        IF nPos_Buffer = 1 GOTO pos_1;
        IF nPos_Buffer = 2 GOTO pos_2;
        IF nPos_Buffer = 3 GOTO pos_3;
        IF nPos_Buffer = 4 GOTO pos_4;
        IF nPos_Buffer = 5 GOTO pos_5;
        IF nPos_Buffer = 6 GOTO pos_6;
        IF nPos_Buffer = 7 GOTO pos_7;
        IF nPos_Buffer = 8 GOTO pos_8;
        IF nPos_Buffer = 9 GOTO pos_9;
        IF nPos_Buffer = 10 GOTO pos_10;
        IF nPos_Buffer = 11 GOTO pos_11;
        IF nPos_Buffer = 12 GOTO pos_12;
        IF nPos_Buffer = 13 GOTO pos_13;
        IF nPos_Buffer = 14 GOTO pos_14;
        IF nPos_Buffer = 15 GOTO pos_15;
        IF nPos_Buffer = 16 GOTO pos_16;
        IF nPos_Buffer = 17 GOTO pos_17;
        IF nPos_Buffer = 18 GOTO pos_18;
        IF nPos_Buffer = 19 GOTO pos_19;
        IF nPos_Buffer = 20 GOTO pos_20;
        IF nPos_Buffer = 21 GOTO pos_21;
        IF nPos_Buffer = 22 GOTO pos_22;
        IF nPos_Buffer = 23 GOTO pos_23;
        IF nPos_Buffer = 24 GOTO pos_24;
        IF nPos_Buffer = 25 GOTO pos_25;
        IF nPos_Buffer = 26 GOTO pos_26;
        IF nPos_Buffer = 27 GOTO pos_27;
        IF nPos_Buffer = 28 GOTO pos_28;
        IF nPos_Buffer = 29 GOTO pos_29;
        IF nPos_Buffer = 30 GOTO pos_30;
        IF nPos_Buffer = 31 GOTO pos_31;
        IF nPos_Buffer = 32 GOTO pos_32;
        IF nPos_Buffer = 33 GOTO pos_33;
        IF nPos_Buffer = 34 GOTO pos_34;
        IF nPos_Buffer = 35 GOTO pos_35;
        IF nPos_Buffer = 36 GOTO pos_36;
        IF nPos_Buffer = 37 GOTO pos_37;
        IF nPos_Buffer = 38 GOTO pos_38;
        IF nPos_Buffer = 39 GOTO pos_39;
        IF nPos_Buffer = 40 GOTO pos_40;
        IF nPos_Buffer = 41 GOTO pos_41;
        IF nPos_Buffer = 42 GOTO pos_42;
        IF nPos_Buffer = 43 GOTO pos_43;
        IF nPos_Buffer = 44 GOTO pos_44;
        IF nPos_Buffer = 45 GOTO pos_45;
        IF nPos_Buffer = 46 GOTO pos_46;
        IF nPos_Buffer = 47 GOTO pos_47;
        IF nPos_Buffer = 48 GOTO pos_48;
        IF nPos_Buffer = 49 GOTO pos_49;
        IF nPos_Buffer = 50 GOTO pos_50;
        IF nPos_Buffer = 51 GOTO pos_51;
        IF nPos_Buffer = 52 GOTO pos_52;
        IF nPos_Buffer = 53 GOTO pos_53;
        IF nPos_Buffer = 54 GOTO pos_54;
        IF nPos_Buffer = 55 GOTO pos_55;
        IF nPos_Buffer = 56 GOTO pos_56;
        IF nPos_Buffer = 57 GOTO pos_57;
        IF nPos_Buffer = 58 GOTO pos_58;
        IF nPos_Buffer = 59 GOTO pos_59;
        IF nPos_Buffer = 60 GOTO pos_60;
        IF nPos_Buffer = 61 GOTO pos_61;
        IF nPos_Buffer = 62 GOTO pos_62;
        IF nPos_Buffer = 63 GOTO pos_63;
        IF nPos_Buffer = 64 GOTO pos_64;
        IF nPos_Buffer = 65 GOTO pos_65;
        IF nPos_Buffer = 66 GOTO pos_66;
        IF nPos_Buffer = 67 GOTO pos_67;
        IF nPos_Buffer = 68 GOTO pos_68;
        IF nPos_Buffer = 69 GOTO pos_69;
        IF nPos_Buffer = 70 GOTO pos_70;
        IF nPos_Buffer = 71 GOTO pos_71;
        IF nPos_Buffer = 72 GOTO pos_72;
        IF nPos_Buffer = 73 GOTO pos_73;
        IF nPos_Buffer = 74 GOTO pos_74;
        IF nPos_Buffer = 75 GOTO pos_75;
        IF nPos_Buffer = 76 GOTO pos_76;
        IF nPos_Buffer = 77 GOTO pos_77;
        IF nPos_Buffer = 78 GOTO pos_78;
        IF nPos_Buffer = 79 GOTO pos_79;
        IF nPos_Buffer = 80 GOTO pos_80;
        IF nPos_Buffer = 81 GOTO pos_81;
        IF nPos_Buffer = 82 GOTO pos_82;
        IF nPos_Buffer = 83 GOTO pos_83;
        IF nPos_Buffer = 84 GOTO pos_84;
        IF nPos_Buffer = 85 GOTO pos_85;
        IF nPos_Buffer = 86 GOTO pos_86;
        IF nPos_Buffer = 87 GOTO pos_87;
        IF nPos_Buffer = 88 GOTO pos_88;
        IF nPos_Buffer = 89 GOTO pos_89;
        IF nPos_Buffer = 90 GOTO pos_90;
        IF nPos_Buffer = 91 GOTO pos_91;
        IF nPos_Buffer = 92 GOTO pos_92;
        IF nPos_Buffer = 93 GOTO pos_93;
        IF nPos_Buffer = 94 GOTO pos_94;
        IF nPos_Buffer = 95 GOTO pos_95;
        IF nPos_Buffer = 96 GOTO pos_96;
        IF nPos_Buffer = 97 GOTO pos_97;
        IF nPos_Buffer = 98 GOTO pos_98;
        IF nPos_Buffer = 99 GOTO pos_99;

    pos_1:
        !Posição 1

        !Carrega posição correspondente à familia selecionada
        IF GInput (PN_IN_Numero_Familia) = 1 THEN
            pPosição_Final_Buffer := pBuffer_Pos_1_Fam_1;
        ENDIF
        IF GInput (PN_IN_Numero_Familia) = 2 THEN
            pPosição_Final_Buffer := pBuffer_Pos_1_Fam_2;
        ENDIF
        IF GInput (PN_IN_Numero_Familia) = 3 THEN
            pPosição_Final_Buffer := pBuffer_Pos_1_Fam_3;
        ENDIF
        IF GInput (PN_IN_Numero_Familia) = 4 THEN
            pPosição_Final_Buffer := pBuffer_Pos_1_Fam_4;
        ENDIF

        GOTO verifica_passo;

    pos_2:
        !Posição 2

        !Carrega posição correspondente à familia selecionada
        IF GInput (PN_IN_Numero_Familia) = 1 THEN
            pPosição_Final_Buffer := pBuffer_Pos_2_Fam_1;
        ENDIF
        IF GInput (PN_IN_Numero_Familia) = 2 THEN
            pPosição_Final_Buffer := pBuffer_Pos_2_Fam_2;
        ENDIF
        IF GInput (PN_IN_Numero_Familia) = 3 THEN
            pPosição_Final_Buffer := pBuffer_Pos_2_Fam_3;
        ENDIF
        IF GInput (PN_IN_Numero_Familia) = 4 THEN
            pPosição_Final_Buffer := pBuffer_Pos_2_Fam_4;
        ENDIF

        GOTO verifica_passo;

    pos_3:
        !Posição 3

        !Carrega posição correspondente à familia selecionada
        IF GInput (PN_IN_Numero_Familia) = 1 THEN
            pPosição_Final_Buffer := pBuffer_Pos_3_Fam_1;
        ENDIF
        IF GInput (PN_IN_Numero_Familia) = 2 THEN
            pPosição_Final_Buffer := pBuffer_Pos_3_Fam_2;
        ENDIF
        IF GInput (PN_IN_Numero_Familia) = 3 THEN
            pPosição_Final_Buffer := pBuffer_Pos_3_Fam_3;
        ENDIF
        IF GInput (PN_IN_Numero_Familia) = 4 THEN
            pPosição_Final_Buffer := pBuffer_Pos_3_Fam_4;
        ENDIF

        GOTO verifica_passo;

    pos_4:
        !Posição 4

        !Carrega posição correspondente à familia selecionada
        IF GInput (PN_IN_Numero_Familia) = 1 THEN
            pPosição_Final_Buffer := pBuffer_Pos_4_Fam_1;
        ENDIF
        IF GInput (PN_IN_Numero_Familia) = 2 THEN
            pPosição_Final_Buffer := pBuffer_Pos_4_Fam_2;
        ENDIF
        IF GInput (PN_IN_Numero_Familia) = 3 THEN
            pPosição_Final_Buffer := pBuffer_Pos_4_Fam_3;
        ENDIF
        IF GInput (PN_IN_Numero_Familia) = 4 THEN
            pPosição_Final_Buffer := pBuffer_Pos_4_Fam_4;
        ENDIF

        GOTO verifica_passo;

    pos_5:
        !Posição 5

        !Carrega posição correspondente à familia selecionada
        IF GInput (PN_IN_Numero_Familia) = 1 THEN
            pPosição_Final_Buffer := pBuffer_Pos_5_Fam_1;
        ENDIF
        IF GInput (PN_IN_Numero_Familia) = 2 THEN
            pPosição_Final_Buffer := pBuffer_Pos_5_Fam_2;
        ENDIF
        IF GInput (PN_IN_Numero_Familia) = 3 THEN
            pPosição_Final_Buffer := pBuffer_Pos_5_Fam_3;
        ENDIF
        IF GInput (PN_IN_Numero_Familia) = 4 THEN
            pPosição_Final_Buffer := pBuffer_Pos_5_Fam_4;
        ENDIF

        GOTO verifica_passo;

    pos_6:
        !Posição 6

        !Carrega posição correspondente à familia selecionada
        IF GInput (PN_IN_Numero_Familia) = 1 THEN
            pPosição_Final_Buffer := pBuffer_Pos_6_Fam_1;
        ENDIF
        IF GInput (PN_IN_Numero_Familia) = 2 THEN
            pPosição_Final_Buffer := pBuffer_Pos_6_Fam_2;
        ENDIF
        IF GInput (PN_IN_Numero_Familia) = 3 THEN
            pPosição_Final_Buffer := pBuffer_Pos_6_Fam_3;
        ENDIF
        IF GInput (PN_IN_Numero_Familia) = 4 THEN
            pPosição_Final_Buffer := pBuffer_Pos_6_Fam_4;
        ENDIF

        GOTO verifica_passo;

    pos_7:
        !Posição 7

        !Carrega posição correspondente à familia selecionada
        IF GInput (PN_IN_Numero_Familia) = 1 THEN
            pPosição_Final_Buffer := pBuffer_Pos_7_Fam_1;
        ENDIF
        IF GInput (PN_IN_Numero_Familia) = 2 THEN
            pPosição_Final_Buffer := pBuffer_Pos_7_Fam_2;
        ENDIF
        IF GInput (PN_IN_Numero_Familia) = 3 THEN
            pPosição_Final_Buffer := pBuffer_Pos_7_Fam_3;
        ENDIF
        IF GInput (PN_IN_Numero_Familia) = 4 THEN
            pPosição_Final_Buffer := pBuffer_Pos_7_Fam_4;
        ENDIF

        GOTO verifica_passo;

    pos_8:
        !Posição 8

        !Carrega posição correspondente à familia selecionada
        IF GInput (PN_IN_Numero_Familia) = 1 THEN
            pPosição_Final_Buffer := pBuffer_Pos_8_Fam_1;
        ENDIF
        IF GInput (PN_IN_Numero_Familia) = 2 THEN
            pPosição_Final_Buffer := pBuffer_Pos_8_Fam_2;
        ENDIF
        IF GInput (PN_IN_Numero_Familia) = 3 THEN
            pPosição_Final_Buffer := pBuffer_Pos_8_Fam_3;
        ENDIF
        IF GInput (PN_IN_Numero_Familia) = 4 THEN
            pPosição_Final_Buffer := pBuffer_Pos_8_Fam_4;
        ENDIF

        GOTO verifica_passo;

    pos_9:
        !Posição 9

        !Carrega posição correspondente à familia selecionada
        IF GInput (PN_IN_Numero_Familia) = 1 THEN
            pPosição_Final_Buffer := pBuffer_Pos_9_Fam_1;
        ENDIF
        IF GInput (PN_IN_Numero_Familia) = 2 THEN
            pPosição_Final_Buffer := pBuffer_Pos_9_Fam_2;
        ENDIF
        IF GInput (PN_IN_Numero_Familia) = 3 THEN
            pPosição_Final_Buffer := pBuffer_Pos_9_Fam_3;
        ENDIF
        IF GInput (PN_IN_Numero_Familia) = 4 THEN
            pPosição_Final_Buffer := pBuffer_Pos_9_Fam_4;
        ENDIF

        GOTO verifica_passo;

    pos_10:
        !Posição 10

        !Carrega posição correspondente à familia selecionada
        IF GInput (PN_IN_Numero_Familia) = 1 THEN
            pPosição_Final_Buffer := pBuffer_Pos_10_Fam_1;
        ENDIF
        IF GInput (PN_IN_Numero_Familia) = 2 THEN
            pPosição_Final_Buffer := pBuffer_Pos_10_Fam_2;
        ENDIF
        IF GInput (PN_IN_Numero_Familia) = 3 THEN
            pPosição_Final_Buffer := pBuffer_Pos_10_Fam_3;
        ENDIF
        IF GInput (PN_IN_Numero_Familia) = 4 THEN
            pPosição_Final_Buffer := pBuffer_Pos_10_Fam_4;
        ENDIF

        GOTO verifica_passo;

    pos_11:
        !Posição 11

        !Carrega posição correspondente à familia selecionada
        IF GInput (PN_IN_Numero_Familia) = 1 THEN
            pPosição_Final_Buffer := pBuffer_Pos_11_Fam_1;
        ENDIF
        IF GInput (PN_IN_Numero_Familia) = 2 THEN
            pPosição_Final_Buffer := pBuffer_Pos_11_Fam_2;
        ENDIF
        IF GInput (PN_IN_Numero_Familia) = 3 THEN
            pPosição_Final_Buffer := pBuffer_Pos_11_Fam_3;
        ENDIF
        IF GInput (PN_IN_Numero_Familia) = 4 THEN
            pPosição_Final_Buffer := pBuffer_Pos_11_Fam_4;
        ENDIF

        GOTO verifica_passo;

    pos_12:
        !Posição 12

        !Carrega posição correspondente à familia selecionada
        IF GInput (PN_IN_Numero_Familia) = 1 THEN
            pPosição_Final_Buffer := pBuffer_Pos_12_Fam_1;
        ENDIF
        IF GInput (PN_IN_Numero_Familia) = 2 THEN
            pPosição_Final_Buffer := pBuffer_Pos_12_Fam_2;
        ENDIF
        IF GInput (PN_IN_Numero_Familia) = 3 THEN
            pPosição_Final_Buffer := pBuffer_Pos_12_Fam_3;
        ENDIF
        IF GInput (PN_IN_Numero_Familia) = 4 THEN
            pPosição_Final_Buffer := pBuffer_Pos_12_Fam_4;
        ENDIF

        GOTO verifica_passo;

    pos_13:
        !Posição 13

        !Carrega posição correspondente à familia selecionada
        IF GInput (PN_IN_Numero_Familia) = 1 THEN
            pPosição_Final_Buffer := pBuffer_Pos_13_Fam_1;
        ENDIF
        IF GInput (PN_IN_Numero_Familia) = 2 THEN
            pPosição_Final_Buffer := pBuffer_Pos_13_Fam_2;
        ENDIF
        IF GInput (PN_IN_Numero_Familia) = 3 THEN
            pPosição_Final_Buffer := pBuffer_Pos_13_Fam_3;
        ENDIF
        IF GInput (PN_IN_Numero_Familia) = 4 THEN
            pPosição_Final_Buffer := pBuffer_Pos_13_Fam_4;
        ENDIF

        GOTO verifica_passo;

    pos_14:
        !Posição 14

        !Carrega posição correspondente à familia selecionada
        IF GInput (PN_IN_Numero_Familia) = 1 THEN
            pPosição_Final_Buffer := pBuffer_Pos_14_Fam_1;
        ENDIF
        IF GInput (PN_IN_Numero_Familia) = 2 THEN
            pPosição_Final_Buffer := pBuffer_Pos_14_Fam_2;
        ENDIF
        IF GInput (PN_IN_Numero_Familia) = 3 THEN
            pPosição_Final_Buffer := pBuffer_Pos_14_Fam_3;
        ENDIF
        IF GInput (PN_IN_Numero_Familia) = 4 THEN
            pPosição_Final_Buffer := pBuffer_Pos_14_Fam_4;
        ENDIF

        GOTO verifica_passo;

    pos_15:
        !Posição 15

        !Carrega posição correspondente à familia selecionada
        IF GInput (PN_IN_Numero_Familia) = 1 THEN
            pPosição_Final_Buffer := pBuffer_Pos_15_Fam_1;
        ENDIF
        IF GInput (PN_IN_Numero_Familia) = 2 THEN
            pPosição_Final_Buffer := pBuffer_Pos_15_Fam_2;
        ENDIF
        IF GInput (PN_IN_Numero_Familia) = 3 THEN
            pPosição_Final_Buffer := pBuffer_Pos_15_Fam_3;
        ENDIF
        IF GInput (PN_IN_Numero_Familia) = 4 THEN
            pPosição_Final_Buffer := pBuffer_Pos_15_Fam_4;
        ENDIF

        GOTO verifica_passo;

    pos_16:
        !Posição 16

        !Carrega posição correspondente à familia selecionada
        IF GInput (PN_IN_Numero_Familia) = 1 THEN
            pPosição_Final_Buffer := pBuffer_Pos_16_Fam_1;
        ENDIF
        IF GInput (PN_IN_Numero_Familia) = 2 THEN
            pPosição_Final_Buffer := pBuffer_Pos_16_Fam_2;
        ENDIF
        IF GInput (PN_IN_Numero_Familia) = 3 THEN
            pPosição_Final_Buffer := pBuffer_Pos_16_Fam_3;
        ENDIF
        IF GInput (PN_IN_Numero_Familia) = 4 THEN
            pPosição_Final_Buffer := pBuffer_Pos_16_Fam_4;
        ENDIF

        GOTO verifica_passo;

    pos_17:
        !Posição 17

        !Carrega posição correspondente à familia selecionada
        IF GInput (PN_IN_Numero_Familia) = 1 THEN
            pPosição_Final_Buffer := pBuffer_Pos_17_Fam_1;
        ENDIF
        IF GInput (PN_IN_Numero_Familia) = 2 THEN
            pPosição_Final_Buffer := pBuffer_Pos_17_Fam_2;
        ENDIF
        IF GInput (PN_IN_Numero_Familia) = 3 THEN
            pPosição_Final_Buffer := pBuffer_Pos_17_Fam_3;
        ENDIF
        IF GInput (PN_IN_Numero_Familia) = 4 THEN
            pPosição_Final_Buffer := pBuffer_Pos_17_Fam_4;
        ENDIF

        GOTO verifica_passo;

    pos_18:
        !Posição 18

        !Carrega posição correspondente à familia selecionada
        IF GInput (PN_IN_Numero_Familia) = 1 THEN
            pPosição_Final_Buffer := pBuffer_Pos_18_Fam_1;
        ENDIF
        IF GInput (PN_IN_Numero_Familia) = 2 THEN
            pPosição_Final_Buffer := pBuffer_Pos_18_Fam_2;
        ENDIF
        IF GInput (PN_IN_Numero_Familia) = 3 THEN
            pPosição_Final_Buffer := pBuffer_Pos_18_Fam_3;
        ENDIF
        IF GInput (PN_IN_Numero_Familia) = 4 THEN
            pPosição_Final_Buffer := pBuffer_Pos_18_Fam_4;
        ENDIF

        GOTO verifica_passo;

    pos_19:
        !Posição 19

        !Carrega posição correspondente à familia selecionada
        IF GInput (PN_IN_Numero_Familia) = 1 THEN
            pPosição_Final_Buffer := pBuffer_Pos_19_Fam_1;
        ENDIF
        IF GInput (PN_IN_Numero_Familia) = 2 THEN
            pPosição_Final_Buffer := pBuffer_Pos_19_Fam_2;
        ENDIF
        IF GInput (PN_IN_Numero_Familia) = 3 THEN
            pPosição_Final_Buffer := pBuffer_Pos_19_Fam_3;
        ENDIF
        IF GInput (PN_IN_Numero_Familia) = 4 THEN
            pPosição_Final_Buffer := pBuffer_Pos_19_Fam_4;
        ENDIF

        GOTO verifica_passo;

    pos_20:
        !Posição 20

        !Carrega posição correspondente à familia selecionada
        IF GInput (PN_IN_Numero_Familia) = 1 THEN
            pPosição_Final_Buffer := pBuffer_Pos_20_Fam_1;
        ENDIF
        IF GInput (PN_IN_Numero_Familia) = 2 THEN
            pPosição_Final_Buffer := pBuffer_Pos_20_Fam_2;
        ENDIF
        IF GInput (PN_IN_Numero_Familia) = 3 THEN
            pPosição_Final_Buffer := pBuffer_Pos_20_Fam_3;
        ENDIF
        IF GInput (PN_IN_Numero_Familia) = 4 THEN
            pPosição_Final_Buffer := pBuffer_Pos_20_Fam_4;
        ENDIF

        GOTO verifica_passo;

    pos_21:
        !Posição 21

        !Carrega posição correspondente à familia selecionada
        IF GInput (PN_IN_Numero_Familia) = 1 THEN
            pPosição_Final_Buffer := pBuffer_Pos_21_Fam_1;
        ENDIF
        IF GInput (PN_IN_Numero_Familia) = 2 THEN
            pPosição_Final_Buffer := pBuffer_Pos_21_Fam_2;
        ENDIF
        IF GInput (PN_IN_Numero_Familia) = 3 THEN
            pPosição_Final_Buffer := pBuffer_Pos_21_Fam_3;
        ENDIF
        IF GInput (PN_IN_Numero_Familia) = 4 THEN
            pPosição_Final_Buffer := pBuffer_Pos_21_Fam_4;
        ENDIF

        GOTO verifica_passo;

    pos_22:
        !Posição 22

        !Carrega posição correspondente à familia selecionada
        IF GInput (PN_IN_Numero_Familia) = 1 THEN
            pPosição_Final_Buffer := pBuffer_Pos_22_Fam_1;
        ENDIF
        IF GInput (PN_IN_Numero_Familia) = 2 THEN
            pPosição_Final_Buffer := pBuffer_Pos_22_Fam_2;
        ENDIF
        IF GInput (PN_IN_Numero_Familia) = 3 THEN
            pPosição_Final_Buffer := pBuffer_Pos_22_Fam_3;
        ENDIF
        IF GInput (PN_IN_Numero_Familia) = 4 THEN
            pPosição_Final_Buffer := pBuffer_Pos_22_Fam_4;
        ENDIF

        GOTO verifica_passo;

    pos_23:
        !Posição 23

        !Carrega posição correspondente à familia selecionada
        IF GInput (PN_IN_Numero_Familia) = 1 THEN
            pPosição_Final_Buffer := pBuffer_Pos_23_Fam_1;
        ENDIF
        IF GInput (PN_IN_Numero_Familia) = 2 THEN
            pPosição_Final_Buffer := pBuffer_Pos_23_Fam_2;
        ENDIF
        IF GInput (PN_IN_Numero_Familia) = 3 THEN
            pPosição_Final_Buffer := pBuffer_Pos_23_Fam_3;
        ENDIF
        IF GInput (PN_IN_Numero_Familia) = 4 THEN
            pPosição_Final_Buffer := pBuffer_Pos_23_Fam_4;
        ENDIF

        GOTO verifica_passo;

    pos_24:
        !Posição 24

        !Carrega posição correspondente à familia selecionada
        IF GInput (PN_IN_Numero_Familia) = 1 THEN
            pPosição_Final_Buffer := pBuffer_Pos_24_Fam_1;
        ENDIF
        IF GInput (PN_IN_Numero_Familia) = 2 THEN
            pPosição_Final_Buffer := pBuffer_Pos_24_Fam_2;
        ENDIF
        IF GInput (PN_IN_Numero_Familia) = 3 THEN
            pPosição_Final_Buffer := pBuffer_Pos_24_Fam_3;
        ENDIF
        IF GInput (PN_IN_Numero_Familia) = 4 THEN
            pPosição_Final_Buffer := pBuffer_Pos_24_Fam_4;
        ENDIF

        GOTO verifica_passo;

    pos_25:
        !Posição 25

        !Carrega posição correspondente à familia selecionada
        IF GInput (PN_IN_Numero_Familia) = 1 THEN
            pPosição_Final_Buffer := pBuffer_Pos_25_Fam_1;
        ENDIF
        IF GInput (PN_IN_Numero_Familia) = 2 THEN
            pPosição_Final_Buffer := pBuffer_Pos_25_Fam_2;
        ENDIF
        IF GInput (PN_IN_Numero_Familia) = 3 THEN
            pPosição_Final_Buffer := pBuffer_Pos_25_Fam_3;
        ENDIF
        IF GInput (PN_IN_Numero_Familia) = 4 THEN
            pPosição_Final_Buffer := pBuffer_Pos_25_Fam_4;
        ENDIF

        GOTO verifica_passo;

    pos_26:
        !Posição 26

        !Carrega posição correspondente à familia selecionada
        IF GInput (PN_IN_Numero_Familia) = 1 THEN
            pPosição_Final_Buffer := pBuffer_Pos_26_Fam_1;
        ENDIF
        IF GInput (PN_IN_Numero_Familia) = 2 THEN
            pPosição_Final_Buffer := pBuffer_Pos_26_Fam_2;
        ENDIF
        IF GInput (PN_IN_Numero_Familia) = 3 THEN
            pPosição_Final_Buffer := pBuffer_Pos_26_Fam_3;
        ENDIF
        IF GInput (PN_IN_Numero_Familia) = 4 THEN
            pPosição_Final_Buffer := pBuffer_Pos_26_Fam_4;
        ENDIF

        GOTO verifica_passo;

    pos_27:
        !Posição 27

        !Carrega posição correspondente à familia selecionada
        IF GInput (PN_IN_Numero_Familia) = 1 THEN
            pPosição_Final_Buffer := pBuffer_Pos_27_Fam_1;
        ENDIF
        IF GInput (PN_IN_Numero_Familia) = 2 THEN
            pPosição_Final_Buffer := pBuffer_Pos_27_Fam_2;
        ENDIF
        IF GInput (PN_IN_Numero_Familia) = 3 THEN
            pPosição_Final_Buffer := pBuffer_Pos_27_Fam_3;
        ENDIF
        IF GInput (PN_IN_Numero_Familia) = 4 THEN
            pPosição_Final_Buffer := pBuffer_Pos_27_Fam_4;
        ENDIF

        GOTO verifica_passo;

    pos_28:
        !Posição 28

        !Carrega posição correspondente à familia selecionada
        IF GInput (PN_IN_Numero_Familia) = 1 THEN
            pPosição_Final_Buffer := pBuffer_Pos_28_Fam_1;
        ENDIF
        IF GInput (PN_IN_Numero_Familia) = 2 THEN
            pPosição_Final_Buffer := pBuffer_Pos_28_Fam_2;
        ENDIF
        IF GInput (PN_IN_Numero_Familia) = 3 THEN
            pPosição_Final_Buffer := pBuffer_Pos_28_Fam_3;
        ENDIF
        IF GInput (PN_IN_Numero_Familia) = 4 THEN
            pPosição_Final_Buffer := pBuffer_Pos_28_Fam_4;
        ENDIF

        GOTO verifica_passo;

    pos_29:
        !Posição 29

        !Carrega posição correspondente à familia selecionada
        IF GInput (PN_IN_Numero_Familia) = 1 THEN
            pPosição_Final_Buffer := pBuffer_Pos_29_Fam_1;
        ENDIF
        IF GInput (PN_IN_Numero_Familia) = 2 THEN
            pPosição_Final_Buffer := pBuffer_Pos_29_Fam_2;
        ENDIF
        IF GInput (PN_IN_Numero_Familia) = 3 THEN
            pPosição_Final_Buffer := pBuffer_Pos_29_Fam_3;
        ENDIF
        IF GInput (PN_IN_Numero_Familia) = 4 THEN
            pPosição_Final_Buffer := pBuffer_Pos_29_Fam_4;
        ENDIF

        GOTO verifica_passo;

    pos_30:
        !Posição 30

        !Carrega posição correspondente à familia selecionada
        IF GInput (PN_IN_Numero_Familia) = 1 THEN
            pPosição_Final_Buffer := pBuffer_Pos_30_Fam_1;
        ENDIF
        IF GInput (PN_IN_Numero_Familia) = 2 THEN
            pPosição_Final_Buffer := pBuffer_Pos_30_Fam_2;
        ENDIF
        IF GInput (PN_IN_Numero_Familia) = 3 THEN
            pPosição_Final_Buffer := pBuffer_Pos_30_Fam_3;
        ENDIF
        IF GInput (PN_IN_Numero_Familia) = 4 THEN
            pPosição_Final_Buffer := pBuffer_Pos_30_Fam_4;
        ENDIF

        GOTO verifica_passo;

    pos_31:
        !Posição 31

        !Carrega posição correspondente à familia selecionada
        IF GInput (PN_IN_Numero_Familia) = 1 THEN
            pPosição_Final_Buffer := pBuffer_Pos_31_Fam_1;
        ENDIF
        IF GInput (PN_IN_Numero_Familia) = 2 THEN
            pPosição_Final_Buffer := pBuffer_Pos_31_Fam_2;
        ENDIF
        IF GInput (PN_IN_Numero_Familia) = 3 THEN
            pPosição_Final_Buffer := pBuffer_Pos_31_Fam_3;
        ENDIF
        IF GInput (PN_IN_Numero_Familia) = 4 THEN
            pPosição_Final_Buffer := pBuffer_Pos_31_Fam_4;
        ENDIF

        GOTO verifica_passo;

    pos_32:
        !Posição 32

        !Carrega posição correspondente à familia selecionada
        IF GInput (PN_IN_Numero_Familia) = 1 THEN
            pPosição_Final_Buffer := pBuffer_Pos_32_Fam_1;
        ENDIF
        IF GInput (PN_IN_Numero_Familia) = 2 THEN
            pPosição_Final_Buffer := pBuffer_Pos_32_Fam_2;
        ENDIF
        IF GInput (PN_IN_Numero_Familia) = 3 THEN
            pPosição_Final_Buffer := pBuffer_Pos_32_Fam_3;
        ENDIF
        IF GInput (PN_IN_Numero_Familia) = 4 THEN
            pPosição_Final_Buffer := pBuffer_Pos_32_Fam_4;
        ENDIF

        GOTO verifica_passo;

    pos_33:
        !Posição 33

        !Carrega posição correspondente à familia selecionada
        IF GInput (PN_IN_Numero_Familia) = 1 THEN
            pPosição_Final_Buffer := pBuffer_Pos_33_Fam_1;
        ENDIF
        IF GInput (PN_IN_Numero_Familia) = 2 THEN
            pPosição_Final_Buffer := pBuffer_Pos_33_Fam_2;
        ENDIF
        IF GInput (PN_IN_Numero_Familia) = 3 THEN
            pPosição_Final_Buffer := pBuffer_Pos_33_Fam_3;
        ENDIF
        IF GInput (PN_IN_Numero_Familia) = 4 THEN
            pPosição_Final_Buffer := pBuffer_Pos_33_Fam_4;
        ENDIF

        GOTO verifica_passo;

    pos_34:
        !Posição 34

        !Carrega posição correspondente à familia selecionada
        IF GInput (PN_IN_Numero_Familia) = 1 THEN
            pPosição_Final_Buffer := pBuffer_Pos_34_Fam_1;
        ENDIF
        IF GInput (PN_IN_Numero_Familia) = 2 THEN
            pPosição_Final_Buffer := pBuffer_Pos_34_Fam_2;
        ENDIF
        IF GInput (PN_IN_Numero_Familia) = 3 THEN
            pPosição_Final_Buffer := pBuffer_Pos_34_Fam_3;
        ENDIF
        IF GInput (PN_IN_Numero_Familia) = 4 THEN
            pPosição_Final_Buffer := pBuffer_Pos_34_Fam_4;
        ENDIF

        GOTO verifica_passo;

    pos_35:
        !Posição 35

        !Carrega posição correspondente à familia selecionada
        IF GInput (PN_IN_Numero_Familia) = 1 THEN
            pPosição_Final_Buffer := pBuffer_Pos_35_Fam_1;
        ENDIF
        IF GInput (PN_IN_Numero_Familia) = 2 THEN
            pPosição_Final_Buffer := pBuffer_Pos_35_Fam_2;
        ENDIF
        IF GInput (PN_IN_Numero_Familia) = 3 THEN
            pPosição_Final_Buffer := pBuffer_Pos_35_Fam_3;
        ENDIF
        IF GInput (PN_IN_Numero_Familia) = 4 THEN
            pPosição_Final_Buffer := pBuffer_Pos_35_Fam_4;
        ENDIF

        GOTO verifica_passo;

    pos_36:
        !Posição 36

        !Carrega posição correspondente à familia selecionada
        IF GInput (PN_IN_Numero_Familia) = 1 THEN
            pPosição_Final_Buffer := pBuffer_Pos_36_Fam_1;
        ENDIF
        IF GInput (PN_IN_Numero_Familia) = 2 THEN
            pPosição_Final_Buffer := pBuffer_Pos_36_Fam_2;
        ENDIF
        IF GInput (PN_IN_Numero_Familia) = 3 THEN
            pPosição_Final_Buffer := pBuffer_Pos_36_Fam_3;
        ENDIF
        IF GInput (PN_IN_Numero_Familia) = 4 THEN
            pPosição_Final_Buffer := pBuffer_Pos_36_Fam_4;
        ENDIF

        GOTO verifica_passo;

    pos_37:
        !Posição 37

        !Carrega posição correspondente à familia selecionada
        IF GInput (PN_IN_Numero_Familia) = 1 THEN
            pPosição_Final_Buffer := pBuffer_Pos_37_Fam_1;
        ENDIF
        IF GInput (PN_IN_Numero_Familia) = 2 THEN
            pPosição_Final_Buffer := pBuffer_Pos_37_Fam_2;
        ENDIF
        IF GInput (PN_IN_Numero_Familia) = 3 THEN
            pPosição_Final_Buffer := pBuffer_Pos_37_Fam_3;
        ENDIF
        IF GInput (PN_IN_Numero_Familia) = 4 THEN
            pPosição_Final_Buffer := pBuffer_Pos_37_Fam_4;
        ENDIF

        GOTO verifica_passo;

    pos_38:
        !Posição 38

        !Carrega posição correspondente à familia selecionada
        IF GInput (PN_IN_Numero_Familia) = 1 THEN
            pPosição_Final_Buffer := pBuffer_Pos_38_Fam_1;
        ENDIF
        IF GInput (PN_IN_Numero_Familia) = 2 THEN
            pPosição_Final_Buffer := pBuffer_Pos_38_Fam_2;
        ENDIF
        IF GInput (PN_IN_Numero_Familia) = 3 THEN
            pPosição_Final_Buffer := pBuffer_Pos_38_Fam_3;
        ENDIF
        IF GInput (PN_IN_Numero_Familia) = 4 THEN
            pPosição_Final_Buffer := pBuffer_Pos_38_Fam_4;
        ENDIF

        GOTO verifica_passo;

    pos_39:
        !Posição 39

        !Carrega posição correspondente à familia selecionada
        IF GInput (PN_IN_Numero_Familia) = 1 THEN
            pPosição_Final_Buffer := pBuffer_Pos_39_Fam_1;
        ENDIF
        IF GInput (PN_IN_Numero_Familia) = 2 THEN
            pPosição_Final_Buffer := pBuffer_Pos_39_Fam_2;
        ENDIF
        IF GInput (PN_IN_Numero_Familia) = 3 THEN
            pPosição_Final_Buffer := pBuffer_Pos_39_Fam_3;
        ENDIF
        IF GInput (PN_IN_Numero_Familia) = 4 THEN
            pPosição_Final_Buffer := pBuffer_Pos_39_Fam_4;
        ENDIF

        GOTO verifica_passo;

    pos_40:
        !Posição 40

        !Carrega posição correspondente à familia selecionada
        IF GInput (PN_IN_Numero_Familia) = 1 THEN
            pPosição_Final_Buffer := pBuffer_Pos_40_Fam_1;
        ENDIF
        IF GInput (PN_IN_Numero_Familia) = 2 THEN
            pPosição_Final_Buffer := pBuffer_Pos_40_Fam_2;
        ENDIF
        IF GInput (PN_IN_Numero_Familia) = 3 THEN
            pPosição_Final_Buffer := pBuffer_Pos_40_Fam_3;
        ENDIF
        IF GInput (PN_IN_Numero_Familia) = 4 THEN
            pPosição_Final_Buffer := pBuffer_Pos_40_Fam_4;
        ENDIF

        GOTO verifica_passo;

    pos_41:
        !Posição 41

        !Carrega posição correspondente à familia selecionada
        IF GInput (PN_IN_Numero_Familia) = 1 THEN
            pPosição_Final_Buffer := pBuffer_Pos_41_Fam_1;
        ENDIF
        IF GInput (PN_IN_Numero_Familia) = 2 THEN
            pPosição_Final_Buffer := pBuffer_Pos_41_Fam_2;
        ENDIF
        IF GInput (PN_IN_Numero_Familia) = 3 THEN
            pPosição_Final_Buffer := pBuffer_Pos_41_Fam_3;
        ENDIF
        IF GInput (PN_IN_Numero_Familia) = 4 THEN
            pPosição_Final_Buffer := pBuffer_Pos_41_Fam_4;
        ENDIF

        GOTO verifica_passo;

    pos_42:
        !Posição 42

        !Carrega posição correspondente à familia selecionada
        IF GInput (PN_IN_Numero_Familia) = 1 THEN
            pPosição_Final_Buffer := pBuffer_Pos_42_Fam_1;
        ENDIF
        IF GInput (PN_IN_Numero_Familia) = 2 THEN
            pPosição_Final_Buffer := pBuffer_Pos_42_Fam_2;
        ENDIF
        IF GInput (PN_IN_Numero_Familia) = 3 THEN
            pPosição_Final_Buffer := pBuffer_Pos_42_Fam_3;
        ENDIF
        IF GInput (PN_IN_Numero_Familia) = 4 THEN
            pPosição_Final_Buffer := pBuffer_Pos_42_Fam_4;
        ENDIF

        GOTO verifica_passo;

    pos_43:
        !Posição 43

        !Carrega posição correspondente à familia selecionada
        IF GInput (PN_IN_Numero_Familia) = 1 THEN
            pPosição_Final_Buffer := pBuffer_Pos_43_Fam_1;
        ENDIF
        IF GInput (PN_IN_Numero_Familia) = 2 THEN
            pPosição_Final_Buffer := pBuffer_Pos_43_Fam_2;
        ENDIF
        IF GInput (PN_IN_Numero_Familia) = 3 THEN
            pPosição_Final_Buffer := pBuffer_Pos_43_Fam_3;
        ENDIF
        IF GInput (PN_IN_Numero_Familia) = 4 THEN
            pPosição_Final_Buffer := pBuffer_Pos_43_Fam_4;
        ENDIF

        GOTO verifica_passo;

    pos_44:
        !Posição 44

        !Carrega posição correspondente à familia selecionada
        IF GInput (PN_IN_Numero_Familia) = 1 THEN
            pPosição_Final_Buffer := pBuffer_Pos_44_Fam_1;
        ENDIF
        IF GInput (PN_IN_Numero_Familia) = 2 THEN
            pPosição_Final_Buffer := pBuffer_Pos_44_Fam_2;
        ENDIF
        IF GInput (PN_IN_Numero_Familia) = 3 THEN
            pPosição_Final_Buffer := pBuffer_Pos_44_Fam_3;
        ENDIF
        IF GInput (PN_IN_Numero_Familia) = 4 THEN
            pPosição_Final_Buffer := pBuffer_Pos_44_Fam_4;
        ENDIF

        GOTO verifica_passo;

    pos_45:
        !Posição 45

        !Carrega posição correspondente à familia selecionada
        IF GInput (PN_IN_Numero_Familia) = 1 THEN
            pPosição_Final_Buffer := pBuffer_Pos_45_Fam_1;
        ENDIF
        IF GInput (PN_IN_Numero_Familia) = 2 THEN
            pPosição_Final_Buffer := pBuffer_Pos_45_Fam_2;
        ENDIF
        IF GInput (PN_IN_Numero_Familia) = 3 THEN
            pPosição_Final_Buffer := pBuffer_Pos_45_Fam_3;
        ENDIF
        IF GInput (PN_IN_Numero_Familia) = 4 THEN
            pPosição_Final_Buffer := pBuffer_Pos_45_Fam_4;
        ENDIF

        GOTO verifica_passo;

    pos_46:
        !Posição 46

        !Carrega posição correspondente à familia selecionada
        IF GInput (PN_IN_Numero_Familia) = 1 THEN
            pPosição_Final_Buffer := pBuffer_Pos_46_Fam_1;
        ENDIF
        IF GInput (PN_IN_Numero_Familia) = 2 THEN
            pPosição_Final_Buffer := pBuffer_Pos_46_Fam_2;
        ENDIF
        IF GInput (PN_IN_Numero_Familia) = 3 THEN
            pPosição_Final_Buffer := pBuffer_Pos_46_Fam_3;
        ENDIF
        IF GInput (PN_IN_Numero_Familia) = 4 THEN
            pPosição_Final_Buffer := pBuffer_Pos_46_Fam_4;
        ENDIF

        GOTO verifica_passo;

    pos_47:
        !Posição 47

        !Carrega posição correspondente à familia selecionada
        IF GInput (PN_IN_Numero_Familia) = 1 THEN
            pPosição_Final_Buffer := pBuffer_Pos_47_Fam_1;
        ENDIF
        IF GInput (PN_IN_Numero_Familia) = 2 THEN
            pPosição_Final_Buffer := pBuffer_Pos_47_Fam_2;
        ENDIF
        IF GInput (PN_IN_Numero_Familia) = 3 THEN
            pPosição_Final_Buffer := pBuffer_Pos_47_Fam_3;
        ENDIF
        IF GInput (PN_IN_Numero_Familia) = 4 THEN
            pPosição_Final_Buffer := pBuffer_Pos_47_Fam_4;
        ENDIF

        GOTO verifica_passo;

    pos_48:
        !Posição 48

        !Carrega posição correspondente à familia selecionada
        IF GInput (PN_IN_Numero_Familia) = 1 THEN
            pPosição_Final_Buffer := pBuffer_Pos_48_Fam_1;
        ENDIF
        IF GInput (PN_IN_Numero_Familia) = 2 THEN
            pPosição_Final_Buffer := pBuffer_Pos_48_Fam_2;
        ENDIF
        IF GInput (PN_IN_Numero_Familia) = 3 THEN
            pPosição_Final_Buffer := pBuffer_Pos_48_Fam_3;
        ENDIF
        IF GInput (PN_IN_Numero_Familia) = 4 THEN
            pPosição_Final_Buffer := pBuffer_Pos_48_Fam_4;
        ENDIF

        GOTO verifica_passo;

    pos_49:
        !Posição 49

        !Carrega posição correspondente à familia selecionada
        IF GInput (PN_IN_Numero_Familia) = 1 THEN
            pPosição_Final_Buffer := pBuffer_Pos_49_Fam_1;
        ENDIF
        IF GInput (PN_IN_Numero_Familia) = 2 THEN
            pPosição_Final_Buffer := pBuffer_Pos_49_Fam_2;
        ENDIF
        IF GInput (PN_IN_Numero_Familia) = 3 THEN
            pPosição_Final_Buffer := pBuffer_Pos_49_Fam_3;
        ENDIF
        IF GInput (PN_IN_Numero_Familia) = 4 THEN
            pPosição_Final_Buffer := pBuffer_Pos_49_Fam_4;
        ENDIF

        GOTO verifica_passo;

    pos_50:
        !Posição 50

        !Carrega posição correspondente à familia selecionada
        IF GInput (PN_IN_Numero_Familia) = 1 THEN
            pPosição_Final_Buffer := pBuffer_Pos_50_Fam_1;
        ENDIF
        IF GInput (PN_IN_Numero_Familia) = 2 THEN
            pPosição_Final_Buffer := pBuffer_Pos_50_Fam_2;
        ENDIF
        IF GInput (PN_IN_Numero_Familia) = 3 THEN
            pPosição_Final_Buffer := pBuffer_Pos_50_Fam_3;
        ENDIF
        IF GInput (PN_IN_Numero_Familia) = 4 THEN
            pPosição_Final_Buffer := pBuffer_Pos_50_Fam_4;
        ENDIF

        GOTO verifica_passo;

    pos_51:
        !Posição 51

        !Carrega posição correspondente à familia selecionada
        IF GInput (PN_IN_Numero_Familia) = 1 THEN
            pPosição_Final_Buffer := pBuffer_Pos_51_Fam_1;
        ENDIF
        IF GInput (PN_IN_Numero_Familia) = 2 THEN
            pPosição_Final_Buffer := pBuffer_Pos_51_Fam_2;
        ENDIF
        IF GInput (PN_IN_Numero_Familia) = 3 THEN
            pPosição_Final_Buffer := pBuffer_Pos_51_Fam_3;
        ENDIF
        IF GInput (PN_IN_Numero_Familia) = 4 THEN
            pPosição_Final_Buffer := pBuffer_Pos_51_Fam_4;
        ENDIF

        GOTO verifica_passo;

    pos_52:
        !Posição 52

        !Carrega posição correspondente à familia selecionada
        IF GInput (PN_IN_Numero_Familia) = 1 THEN
            pPosição_Final_Buffer := pBuffer_Pos_52_Fam_1;
        ENDIF
        IF GInput (PN_IN_Numero_Familia) = 2 THEN
            pPosição_Final_Buffer := pBuffer_Pos_52_Fam_2;
        ENDIF
        IF GInput (PN_IN_Numero_Familia) = 3 THEN
            pPosição_Final_Buffer := pBuffer_Pos_52_Fam_3;
        ENDIF
        IF GInput (PN_IN_Numero_Familia) = 4 THEN
            pPosição_Final_Buffer := pBuffer_Pos_52_Fam_4;
        ENDIF

        GOTO verifica_passo;

    pos_53:
        !Posição 53

        !Carrega posição correspondente à familia selecionada
        IF GInput (PN_IN_Numero_Familia) = 1 THEN
            pPosição_Final_Buffer := pBuffer_Pos_53_Fam_1;
        ENDIF
        IF GInput (PN_IN_Numero_Familia) = 2 THEN
            pPosição_Final_Buffer := pBuffer_Pos_53_Fam_2;
        ENDIF
        IF GInput (PN_IN_Numero_Familia) = 3 THEN
            pPosição_Final_Buffer := pBuffer_Pos_53_Fam_3;
        ENDIF
        IF GInput (PN_IN_Numero_Familia) = 4 THEN
            pPosição_Final_Buffer := pBuffer_Pos_53_Fam_4;
        ENDIF

        GOTO verifica_passo;

    pos_54:
        !Posição 54

        !Carrega posição correspondente à familia selecionada
        IF GInput (PN_IN_Numero_Familia) = 1 THEN
            pPosição_Final_Buffer := pBuffer_Pos_54_Fam_1;
        ENDIF
        IF GInput (PN_IN_Numero_Familia) = 2 THEN
            pPosição_Final_Buffer := pBuffer_Pos_54_Fam_2;
        ENDIF
        IF GInput (PN_IN_Numero_Familia) = 3 THEN
            pPosição_Final_Buffer := pBuffer_Pos_54_Fam_3;
        ENDIF
        IF GInput (PN_IN_Numero_Familia) = 4 THEN
            pPosição_Final_Buffer := pBuffer_Pos_54_Fam_4;
        ENDIF

        GOTO verifica_passo;

    pos_55:
        !Posição 55

        !Carrega posição correspondente à familia selecionada
        IF GInput (PN_IN_Numero_Familia) = 1 THEN
            pPosição_Final_Buffer := pBuffer_Pos_55_Fam_1;
        ENDIF
        IF GInput (PN_IN_Numero_Familia) = 2 THEN
            pPosição_Final_Buffer := pBuffer_Pos_55_Fam_2;
        ENDIF
        IF GInput (PN_IN_Numero_Familia) = 3 THEN
            pPosição_Final_Buffer := pBuffer_Pos_55_Fam_3;
        ENDIF
        IF GInput (PN_IN_Numero_Familia) = 4 THEN
            pPosição_Final_Buffer := pBuffer_Pos_55_Fam_4;
        ENDIF

        GOTO verifica_passo;

    pos_56:
        !Posição 56

        !Carrega posição correspondente à familia selecionada
        IF GInput (PN_IN_Numero_Familia) = 1 THEN
            pPosição_Final_Buffer := pBuffer_Pos_56_Fam_1;
        ENDIF
        IF GInput (PN_IN_Numero_Familia) = 2 THEN
            pPosição_Final_Buffer := pBuffer_Pos_56_Fam_2;
        ENDIF
        IF GInput (PN_IN_Numero_Familia) = 3 THEN
            pPosição_Final_Buffer := pBuffer_Pos_56_Fam_3;
        ENDIF
        IF GInput (PN_IN_Numero_Familia) = 4 THEN
            pPosição_Final_Buffer := pBuffer_Pos_56_Fam_4;
        ENDIF

        GOTO verifica_passo;

    pos_57:
        !Posição 57

        !Carrega posição correspondente à familia selecionada
        IF GInput (PN_IN_Numero_Familia) = 1 THEN
            pPosição_Final_Buffer := pBuffer_Pos_57_Fam_1;
        ENDIF
        IF GInput (PN_IN_Numero_Familia) = 2 THEN
            pPosição_Final_Buffer := pBuffer_Pos_57_Fam_2;
        ENDIF
        IF GInput (PN_IN_Numero_Familia) = 3 THEN
            pPosição_Final_Buffer := pBuffer_Pos_57_Fam_3;
        ENDIF
        IF GInput (PN_IN_Numero_Familia) = 4 THEN
            pPosição_Final_Buffer := pBuffer_Pos_57_Fam_4;
        ENDIF

        GOTO verifica_passo;

    pos_58:
        !Posição 58

        !Carrega posição correspondente à familia selecionada
        IF GInput (PN_IN_Numero_Familia) = 1 THEN
            pPosição_Final_Buffer := pBuffer_Pos_58_Fam_1;
        ENDIF
        IF GInput (PN_IN_Numero_Familia) = 2 THEN
            pPosição_Final_Buffer := pBuffer_Pos_58_Fam_2;
        ENDIF
        IF GInput (PN_IN_Numero_Familia) = 3 THEN
            pPosição_Final_Buffer := pBuffer_Pos_58_Fam_3;
        ENDIF
        IF GInput (PN_IN_Numero_Familia) = 4 THEN
            pPosição_Final_Buffer := pBuffer_Pos_58_Fam_4;
        ENDIF

        GOTO verifica_passo;

    pos_59:
        !Posição 59

        !Carrega posição correspondente à familia selecionada
        IF GInput (PN_IN_Numero_Familia) = 1 THEN
            pPosição_Final_Buffer := pBuffer_Pos_59_Fam_1;
        ENDIF
        IF GInput (PN_IN_Numero_Familia) = 2 THEN
            pPosição_Final_Buffer := pBuffer_Pos_59_Fam_2;
        ENDIF
        IF GInput (PN_IN_Numero_Familia) = 3 THEN
            pPosição_Final_Buffer := pBuffer_Pos_59_Fam_3;
        ENDIF
        IF GInput (PN_IN_Numero_Familia) = 4 THEN
            pPosição_Final_Buffer := pBuffer_Pos_59_Fam_4;
        ENDIF

        GOTO verifica_passo;

    pos_60:
        !Posição 60

        !Carrega posição correspondente à familia selecionada
        IF GInput (PN_IN_Numero_Familia) = 1 THEN
            pPosição_Final_Buffer := pBuffer_Pos_60_Fam_1;
        ENDIF
        IF GInput (PN_IN_Numero_Familia) = 2 THEN
            pPosição_Final_Buffer := pBuffer_Pos_60_Fam_2;
        ENDIF
        IF GInput (PN_IN_Numero_Familia) = 3 THEN
            pPosição_Final_Buffer := pBuffer_Pos_60_Fam_3;
        ENDIF
        IF GInput (PN_IN_Numero_Familia) = 4 THEN
            pPosição_Final_Buffer := pBuffer_Pos_60_Fam_4;
        ENDIF

        GOTO verifica_passo;

    pos_61:
        !Posição 61

        !Carrega posição correspondente à familia selecionada
        IF GInput (PN_IN_Numero_Familia) = 1 THEN
            pPosição_Final_Buffer := pBuffer_Pos_61_Fam_1;
        ENDIF
        IF GInput (PN_IN_Numero_Familia) = 2 THEN
            pPosição_Final_Buffer := pBuffer_Pos_61_Fam_2;
        ENDIF
        IF GInput (PN_IN_Numero_Familia) = 3 THEN
            pPosição_Final_Buffer := pBuffer_Pos_61_Fam_3;
        ENDIF
        IF GInput (PN_IN_Numero_Familia) = 4 THEN
            pPosição_Final_Buffer := pBuffer_Pos_61_Fam_4;
        ENDIF

        GOTO verifica_passo;

    pos_62:
        !Posição 62

        !Carrega posição correspondente à familia selecionada
        IF GInput (PN_IN_Numero_Familia) = 1 THEN
            pPosição_Final_Buffer := pBuffer_Pos_62_Fam_1;
        ENDIF
        IF GInput (PN_IN_Numero_Familia) = 2 THEN
            pPosição_Final_Buffer := pBuffer_Pos_62_Fam_2;
        ENDIF
        IF GInput (PN_IN_Numero_Familia) = 3 THEN
            pPosição_Final_Buffer := pBuffer_Pos_62_Fam_3;
        ENDIF
        IF GInput (PN_IN_Numero_Familia) = 4 THEN
            pPosição_Final_Buffer := pBuffer_Pos_62_Fam_4;
        ENDIF

        GOTO verifica_passo;

    pos_63:
        !Posição 63

        !Carrega posição correspondente à familia selecionada
        IF GInput (PN_IN_Numero_Familia) = 1 THEN
            pPosição_Final_Buffer := pBuffer_Pos_63_Fam_1;
        ENDIF
        IF GInput (PN_IN_Numero_Familia) = 2 THEN
            pPosição_Final_Buffer := pBuffer_Pos_63_Fam_2;
        ENDIF
        IF GInput (PN_IN_Numero_Familia) = 3 THEN
            pPosição_Final_Buffer := pBuffer_Pos_63_Fam_3;
        ENDIF
        IF GInput (PN_IN_Numero_Familia) = 4 THEN
            pPosição_Final_Buffer := pBuffer_Pos_63_Fam_4;
        ENDIF

        GOTO verifica_passo;

    pos_64:
        !Posição 64

        !Carrega posição correspondente à familia selecionada
        IF GInput (PN_IN_Numero_Familia) = 1 THEN
            pPosição_Final_Buffer := pBuffer_Pos_64_Fam_1;
        ENDIF
        IF GInput (PN_IN_Numero_Familia) = 2 THEN
            pPosição_Final_Buffer := pBuffer_Pos_64_Fam_2;
        ENDIF
        IF GInput (PN_IN_Numero_Familia) = 3 THEN
            pPosição_Final_Buffer := pBuffer_Pos_64_Fam_3;
        ENDIF
        IF GInput (PN_IN_Numero_Familia) = 4 THEN
            pPosição_Final_Buffer := pBuffer_Pos_64_Fam_4;
        ENDIF

        GOTO verifica_passo;

    pos_65:
        !Posição 65

        !Carrega posição correspondente à familia selecionada
        IF GInput (PN_IN_Numero_Familia) = 1 THEN
            pPosição_Final_Buffer := pBuffer_Pos_65_Fam_1;
        ENDIF
        IF GInput (PN_IN_Numero_Familia) = 2 THEN
            pPosição_Final_Buffer := pBuffer_Pos_65_Fam_2;
        ENDIF
        IF GInput (PN_IN_Numero_Familia) = 3 THEN
            pPosição_Final_Buffer := pBuffer_Pos_65_Fam_3;
        ENDIF
        IF GInput (PN_IN_Numero_Familia) = 4 THEN
            pPosição_Final_Buffer := pBuffer_Pos_65_Fam_4;
        ENDIF

        GOTO verifica_passo;

    pos_66:
        !Posição 66

        !Carrega posição correspondente à familia selecionada
        IF GInput (PN_IN_Numero_Familia) = 1 THEN
            pPosição_Final_Buffer := pBuffer_Pos_66_Fam_1;
        ENDIF
        IF GInput (PN_IN_Numero_Familia) = 2 THEN
            pPosição_Final_Buffer := pBuffer_Pos_66_Fam_2;
        ENDIF
        IF GInput (PN_IN_Numero_Familia) = 3 THEN
            pPosição_Final_Buffer := pBuffer_Pos_66_Fam_3;
        ENDIF
        IF GInput (PN_IN_Numero_Familia) = 4 THEN
            pPosição_Final_Buffer := pBuffer_Pos_66_Fam_4;
        ENDIF

        GOTO verifica_passo;

    pos_67:
        !Posição 67

        !Carrega posição correspondente à familia selecionada
        IF GInput (PN_IN_Numero_Familia) = 1 THEN
            pPosição_Final_Buffer := pBuffer_Pos_67_Fam_1;
        ENDIF
        IF GInput (PN_IN_Numero_Familia) = 2 THEN
            pPosição_Final_Buffer := pBuffer_Pos_67_Fam_2;
        ENDIF
        IF GInput (PN_IN_Numero_Familia) = 3 THEN
            pPosição_Final_Buffer := pBuffer_Pos_67_Fam_3;
        ENDIF
        IF GInput (PN_IN_Numero_Familia) = 4 THEN
            pPosição_Final_Buffer := pBuffer_Pos_67_Fam_4;
        ENDIF

        GOTO verifica_passo;

    pos_68:
        !Posição 68

        !Carrega posição correspondente à familia selecionada
        IF GInput (PN_IN_Numero_Familia) = 1 THEN
            pPosição_Final_Buffer := pBuffer_Pos_68_Fam_1;
        ENDIF
        IF GInput (PN_IN_Numero_Familia) = 2 THEN
            pPosição_Final_Buffer := pBuffer_Pos_68_Fam_2;
        ENDIF
        IF GInput (PN_IN_Numero_Familia) = 3 THEN
            pPosição_Final_Buffer := pBuffer_Pos_68_Fam_3;
        ENDIF
        IF GInput (PN_IN_Numero_Familia) = 4 THEN
            pPosição_Final_Buffer := pBuffer_Pos_68_Fam_4;
        ENDIF

        GOTO verifica_passo;

    pos_69:
        !Posição 69

        !Carrega posição correspondente à familia selecionada
        IF GInput (PN_IN_Numero_Familia) = 1 THEN
            pPosição_Final_Buffer := pBuffer_Pos_69_Fam_1;
        ENDIF
        IF GInput (PN_IN_Numero_Familia) = 2 THEN
            pPosição_Final_Buffer := pBuffer_Pos_69_Fam_2;
        ENDIF
        IF GInput (PN_IN_Numero_Familia) = 3 THEN
            pPosição_Final_Buffer := pBuffer_Pos_69_Fam_3;
        ENDIF
        IF GInput (PN_IN_Numero_Familia) = 4 THEN
            pPosição_Final_Buffer := pBuffer_Pos_69_Fam_4;
        ENDIF

        GOTO verifica_passo;

    pos_70:
        !Posição 70

        !Carrega posição correspondente à familia selecionada
        IF GInput (PN_IN_Numero_Familia) = 1 THEN
            pPosição_Final_Buffer := pBuffer_Pos_70_Fam_1;
        ENDIF
        IF GInput (PN_IN_Numero_Familia) = 2 THEN
            pPosição_Final_Buffer := pBuffer_Pos_70_Fam_2;
        ENDIF
        IF GInput (PN_IN_Numero_Familia) = 3 THEN
            pPosição_Final_Buffer := pBuffer_Pos_70_Fam_3;
        ENDIF
        IF GInput (PN_IN_Numero_Familia) = 4 THEN
            pPosição_Final_Buffer := pBuffer_Pos_70_Fam_4;
        ENDIF

        GOTO verifica_passo;

    pos_71:
        !Posição 71

        !Carrega posição correspondente à familia selecionada
        IF GInput (PN_IN_Numero_Familia) = 1 THEN
            pPosição_Final_Buffer := pBuffer_Pos_71_Fam_1;
        ENDIF
        IF GInput (PN_IN_Numero_Familia) = 2 THEN
            pPosição_Final_Buffer := pBuffer_Pos_71_Fam_2;
        ENDIF
        IF GInput (PN_IN_Numero_Familia) = 3 THEN
            pPosição_Final_Buffer := pBuffer_Pos_71_Fam_3;
        ENDIF
        IF GInput (PN_IN_Numero_Familia) = 4 THEN
            pPosição_Final_Buffer := pBuffer_Pos_71_Fam_4;
        ENDIF

        GOTO verifica_passo;

    pos_72:
        !Posição 72

        !Carrega posição correspondente à familia selecionada
        IF GInput (PN_IN_Numero_Familia) = 1 THEN
            pPosição_Final_Buffer := pBuffer_Pos_72_Fam_1;
        ENDIF
        IF GInput (PN_IN_Numero_Familia) = 2 THEN
            pPosição_Final_Buffer := pBuffer_Pos_72_Fam_2;
        ENDIF
        IF GInput (PN_IN_Numero_Familia) = 3 THEN
            pPosição_Final_Buffer := pBuffer_Pos_72_Fam_3;
        ENDIF
        IF GInput (PN_IN_Numero_Familia) = 4 THEN
            pPosição_Final_Buffer := pBuffer_Pos_72_Fam_4;
        ENDIF

        GOTO verifica_passo;

    pos_73:
        !Posição 73

        !Carrega posição correspondente à familia selecionada
        IF GInput (PN_IN_Numero_Familia) = 1 THEN
            pPosição_Final_Buffer := pBuffer_Pos_73_Fam_1;
        ENDIF
        IF GInput (PN_IN_Numero_Familia) = 2 THEN
            pPosição_Final_Buffer := pBuffer_Pos_73_Fam_2;
        ENDIF
        IF GInput (PN_IN_Numero_Familia) = 3 THEN
            pPosição_Final_Buffer := pBuffer_Pos_73_Fam_3;
        ENDIF
        IF GInput (PN_IN_Numero_Familia) = 4 THEN
            pPosição_Final_Buffer := pBuffer_Pos_73_Fam_4;
        ENDIF

        GOTO verifica_passo;

    pos_74:
        !Posição 74

        !Carrega posição correspondente à familia selecionada
        IF GInput (PN_IN_Numero_Familia) = 1 THEN
            pPosição_Final_Buffer := pBuffer_Pos_74_Fam_1;
        ENDIF
        IF GInput (PN_IN_Numero_Familia) = 2 THEN
            pPosição_Final_Buffer := pBuffer_Pos_74_Fam_2;
        ENDIF
        IF GInput (PN_IN_Numero_Familia) = 3 THEN
            pPosição_Final_Buffer := pBuffer_Pos_74_Fam_3;
        ENDIF
        IF GInput (PN_IN_Numero_Familia) = 4 THEN
            pPosição_Final_Buffer := pBuffer_Pos_74_Fam_4;
        ENDIF

        GOTO verifica_passo;

    pos_75:
        !Posição 75

        !Carrega posição correspondente à familia selecionada
        IF GInput (PN_IN_Numero_Familia) = 1 THEN
            pPosição_Final_Buffer := pBuffer_Pos_75_Fam_1;
        ENDIF
        IF GInput (PN_IN_Numero_Familia) = 2 THEN
            pPosição_Final_Buffer := pBuffer_Pos_75_Fam_2;
        ENDIF
        IF GInput (PN_IN_Numero_Familia) = 3 THEN
            pPosição_Final_Buffer := pBuffer_Pos_75_Fam_3;
        ENDIF
        IF GInput (PN_IN_Numero_Familia) = 4 THEN
            pPosição_Final_Buffer := pBuffer_Pos_75_Fam_4;
        ENDIF

        GOTO verifica_passo;

    pos_76:
        !Posição 76

        !Carrega posição correspondente à familia selecionada
        IF GInput (PN_IN_Numero_Familia) = 1 THEN
            pPosição_Final_Buffer := pBuffer_Pos_76_Fam_1;
        ENDIF
        IF GInput (PN_IN_Numero_Familia) = 2 THEN
            pPosição_Final_Buffer := pBuffer_Pos_76_Fam_2;
        ENDIF
        IF GInput (PN_IN_Numero_Familia) = 3 THEN
            pPosição_Final_Buffer := pBuffer_Pos_76_Fam_3;
        ENDIF
        IF GInput (PN_IN_Numero_Familia) = 4 THEN
            pPosição_Final_Buffer := pBuffer_Pos_76_Fam_4;
        ENDIF

        GOTO verifica_passo;

    pos_77:
        !Posição 77

        !Carrega posição correspondente à familia selecionada
        IF GInput (PN_IN_Numero_Familia) = 1 THEN
            pPosição_Final_Buffer := pBuffer_Pos_77_Fam_1;
        ENDIF
        IF GInput (PN_IN_Numero_Familia) = 2 THEN
            pPosição_Final_Buffer := pBuffer_Pos_77_Fam_2;
        ENDIF
        IF GInput (PN_IN_Numero_Familia) = 3 THEN
            pPosição_Final_Buffer := pBuffer_Pos_77_Fam_3;
        ENDIF
        IF GInput (PN_IN_Numero_Familia) = 4 THEN
            pPosição_Final_Buffer := pBuffer_Pos_77_Fam_4;
        ENDIF

        GOTO verifica_passo;

    pos_78:
        !Posição 78

        !Carrega posição correspondente à familia selecionada
        IF GInput (PN_IN_Numero_Familia) = 1 THEN
            pPosição_Final_Buffer := pBuffer_Pos_78_Fam_1;
        ENDIF
        IF GInput (PN_IN_Numero_Familia) = 2 THEN
            pPosição_Final_Buffer := pBuffer_Pos_78_Fam_2;
        ENDIF
        IF GInput (PN_IN_Numero_Familia) = 3 THEN
            pPosição_Final_Buffer := pBuffer_Pos_78_Fam_3;
        ENDIF
        IF GInput (PN_IN_Numero_Familia) = 4 THEN
            pPosição_Final_Buffer := pBuffer_Pos_78_Fam_4;
        ENDIF

        GOTO verifica_passo;

    pos_79:
        !Posição 79

        !Carrega posição correspondente à familia selecionada
        IF GInput (PN_IN_Numero_Familia) = 1 THEN
            pPosição_Final_Buffer := pBuffer_Pos_79_Fam_1;
        ENDIF
        IF GInput (PN_IN_Numero_Familia) = 2 THEN
            pPosição_Final_Buffer := pBuffer_Pos_79_Fam_2;
        ENDIF
        IF GInput (PN_IN_Numero_Familia) = 3 THEN
            pPosição_Final_Buffer := pBuffer_Pos_79_Fam_3;
        ENDIF
        IF GInput (PN_IN_Numero_Familia) = 4 THEN
            pPosição_Final_Buffer := pBuffer_Pos_79_Fam_4;
        ENDIF

        GOTO verifica_passo;

    pos_80:
        !Posição 80

        !Carrega posição correspondente à familia selecionada
        IF GInput (PN_IN_Numero_Familia) = 1 THEN
            pPosição_Final_Buffer := pBuffer_Pos_80_Fam_1;
        ENDIF
        IF GInput (PN_IN_Numero_Familia) = 2 THEN
            pPosição_Final_Buffer := pBuffer_Pos_80_Fam_2;
        ENDIF
        IF GInput (PN_IN_Numero_Familia) = 3 THEN
            pPosição_Final_Buffer := pBuffer_Pos_80_Fam_3;
        ENDIF
        IF GInput (PN_IN_Numero_Familia) = 4 THEN
            pPosição_Final_Buffer := pBuffer_Pos_80_Fam_4;
        ENDIF

        GOTO verifica_passo;

    pos_81:
        !Posição 81

        !Carrega posição correspondente à familia selecionada
        IF GInput (PN_IN_Numero_Familia) = 1 THEN
            pPosição_Final_Buffer := pBuffer_Pos_81_Fam_1;
        ENDIF
        IF GInput (PN_IN_Numero_Familia) = 2 THEN
            pPosição_Final_Buffer := pBuffer_Pos_81_Fam_2;
        ENDIF
        IF GInput (PN_IN_Numero_Familia) = 3 THEN
            pPosição_Final_Buffer := pBuffer_Pos_81_Fam_3;
        ENDIF
        IF GInput (PN_IN_Numero_Familia) = 4 THEN
            pPosição_Final_Buffer := pBuffer_Pos_81_Fam_4;
        ENDIF

        GOTO verifica_passo;

    pos_82:
        !Posição 82

        !Carrega posição correspondente à familia selecionada
        IF GInput (PN_IN_Numero_Familia) = 1 THEN
            pPosição_Final_Buffer := pBuffer_Pos_82_Fam_1;
        ENDIF
        IF GInput (PN_IN_Numero_Familia) = 2 THEN
            pPosição_Final_Buffer := pBuffer_Pos_82_Fam_2;
        ENDIF
        IF GInput (PN_IN_Numero_Familia) = 3 THEN
            pPosição_Final_Buffer := pBuffer_Pos_82_Fam_3;
        ENDIF
        IF GInput (PN_IN_Numero_Familia) = 4 THEN
            pPosição_Final_Buffer := pBuffer_Pos_82_Fam_4;
        ENDIF

        GOTO verifica_passo;

    pos_83:
        !Posição 83

        !Carrega posição correspondente à familia selecionada
        IF GInput (PN_IN_Numero_Familia) = 1 THEN
            pPosição_Final_Buffer := pBuffer_Pos_83_Fam_1;
        ENDIF
        IF GInput (PN_IN_Numero_Familia) = 2 THEN
            pPosição_Final_Buffer := pBuffer_Pos_83_Fam_2;
        ENDIF
        IF GInput (PN_IN_Numero_Familia) = 3 THEN
            pPosição_Final_Buffer := pBuffer_Pos_83_Fam_3;
        ENDIF
        IF GInput (PN_IN_Numero_Familia) = 4 THEN
            pPosição_Final_Buffer := pBuffer_Pos_83_Fam_4;
        ENDIF

        GOTO verifica_passo;

    pos_84:
        !Posição 84

        !Carrega posição correspondente à familia selecionada
        IF GInput (PN_IN_Numero_Familia) = 1 THEN
            pPosição_Final_Buffer := pBuffer_Pos_84_Fam_1;
        ENDIF
        IF GInput (PN_IN_Numero_Familia) = 2 THEN
            pPosição_Final_Buffer := pBuffer_Pos_84_Fam_2;
        ENDIF
        IF GInput (PN_IN_Numero_Familia) = 3 THEN
            pPosição_Final_Buffer := pBuffer_Pos_84_Fam_3;
        ENDIF
        IF GInput (PN_IN_Numero_Familia) = 4 THEN
            pPosição_Final_Buffer := pBuffer_Pos_84_Fam_4;
        ENDIF

        GOTO verifica_passo;

    pos_85:
        !Posição 85

        !Carrega posição correspondente à familia selecionada
        IF GInput (PN_IN_Numero_Familia) = 1 THEN
            pPosição_Final_Buffer := pBuffer_Pos_85_Fam_1;
        ENDIF
        IF GInput (PN_IN_Numero_Familia) = 2 THEN
            pPosição_Final_Buffer := pBuffer_Pos_85_Fam_2;
        ENDIF
        IF GInput (PN_IN_Numero_Familia) = 3 THEN
            pPosição_Final_Buffer := pBuffer_Pos_85_Fam_3;
        ENDIF
        IF GInput (PN_IN_Numero_Familia) = 4 THEN
            pPosição_Final_Buffer := pBuffer_Pos_85_Fam_4;
        ENDIF

        GOTO verifica_passo;

    pos_86:
        !Posição 86

        !Carrega posição correspondente à familia selecionada
        IF GInput (PN_IN_Numero_Familia) = 1 THEN
            pPosição_Final_Buffer := pBuffer_Pos_86_Fam_1;
        ENDIF
        IF GInput (PN_IN_Numero_Familia) = 2 THEN
            pPosição_Final_Buffer := pBuffer_Pos_86_Fam_2;
        ENDIF
        IF GInput (PN_IN_Numero_Familia) = 3 THEN
            pPosição_Final_Buffer := pBuffer_Pos_86_Fam_3;
        ENDIF
        IF GInput (PN_IN_Numero_Familia) = 4 THEN
            pPosição_Final_Buffer := pBuffer_Pos_86_Fam_4;
        ENDIF

        GOTO verifica_passo;

    pos_87:
        !Posição 87

        !Carrega posição correspondente à familia selecionada
        IF GInput (PN_IN_Numero_Familia) = 1 THEN
            pPosição_Final_Buffer := pBuffer_Pos_87_Fam_1;
        ENDIF
        IF GInput (PN_IN_Numero_Familia) = 2 THEN
            pPosição_Final_Buffer := pBuffer_Pos_87_Fam_2;
        ENDIF
        IF GInput (PN_IN_Numero_Familia) = 3 THEN
            pPosição_Final_Buffer := pBuffer_Pos_87_Fam_3;
        ENDIF
        IF GInput (PN_IN_Numero_Familia) = 4 THEN
            pPosição_Final_Buffer := pBuffer_Pos_87_Fam_4;
        ENDIF

        GOTO verifica_passo;

    pos_88:
        !Posição 88

        !Carrega posição correspondente à familia selecionada
        IF GInput (PN_IN_Numero_Familia) = 1 THEN
            pPosição_Final_Buffer := pBuffer_Pos_88_Fam_1;
        ENDIF
        IF GInput (PN_IN_Numero_Familia) = 2 THEN
            pPosição_Final_Buffer := pBuffer_Pos_88_Fam_2;
        ENDIF
        IF GInput (PN_IN_Numero_Familia) = 3 THEN
            pPosição_Final_Buffer := pBuffer_Pos_88_Fam_3;
        ENDIF
        IF GInput (PN_IN_Numero_Familia) = 4 THEN
            pPosição_Final_Buffer := pBuffer_Pos_88_Fam_4;
        ENDIF

        GOTO verifica_passo;

    pos_89:
        !Posição 89

        !Carrega posição correspondente à familia selecionada
        IF GInput (PN_IN_Numero_Familia) = 1 THEN
            pPosição_Final_Buffer := pBuffer_Pos_89_Fam_1;
        ENDIF
        IF GInput (PN_IN_Numero_Familia) = 2 THEN
            pPosição_Final_Buffer := pBuffer_Pos_89_Fam_2;
        ENDIF
        IF GInput (PN_IN_Numero_Familia) = 3 THEN
            pPosição_Final_Buffer := pBuffer_Pos_89_Fam_3;
        ENDIF
        IF GInput (PN_IN_Numero_Familia) = 4 THEN
            pPosição_Final_Buffer := pBuffer_Pos_89_Fam_4;
        ENDIF

        GOTO verifica_passo;

    pos_90:
        !Posição 90

        !Carrega posição correspondente à familia selecionada
        IF GInput (PN_IN_Numero_Familia) = 1 THEN
            pPosição_Final_Buffer := pBuffer_Pos_90_Fam_1;
        ENDIF
        IF GInput (PN_IN_Numero_Familia) = 2 THEN
            pPosição_Final_Buffer := pBuffer_Pos_90_Fam_2;
        ENDIF
        IF GInput (PN_IN_Numero_Familia) = 3 THEN
            pPosição_Final_Buffer := pBuffer_Pos_90_Fam_3;
        ENDIF
        IF GInput (PN_IN_Numero_Familia) = 4 THEN
            pPosição_Final_Buffer := pBuffer_Pos_90_Fam_4;
        ENDIF

        GOTO verifica_passo;

    pos_91:
        !Posição 91

        !Carrega posição correspondente à familia selecionada
        IF GInput (PN_IN_Numero_Familia) = 1 THEN
            pPosição_Final_Buffer := pBuffer_Pos_91_Fam_1;
        ENDIF
        IF GInput (PN_IN_Numero_Familia) = 2 THEN
            pPosição_Final_Buffer := pBuffer_Pos_91_Fam_2;
        ENDIF
        IF GInput (PN_IN_Numero_Familia) = 3 THEN
            pPosição_Final_Buffer := pBuffer_Pos_91_Fam_3;
        ENDIF
        IF GInput (PN_IN_Numero_Familia) = 4 THEN
            pPosição_Final_Buffer := pBuffer_Pos_91_Fam_4;
        ENDIF

        GOTO verifica_passo;

    pos_92:
        !Posição 92

        !Carrega posição correspondente à familia selecionada
        IF GInput (PN_IN_Numero_Familia) = 1 THEN
            pPosição_Final_Buffer := pBuffer_Pos_92_Fam_1;
        ENDIF
        IF GInput (PN_IN_Numero_Familia) = 2 THEN
            pPosição_Final_Buffer := pBuffer_Pos_92_Fam_2;
        ENDIF
        IF GInput (PN_IN_Numero_Familia) = 3 THEN
            pPosição_Final_Buffer := pBuffer_Pos_92_Fam_3;
        ENDIF
        IF GInput (PN_IN_Numero_Familia) = 4 THEN
            pPosição_Final_Buffer := pBuffer_Pos_92_Fam_4;
        ENDIF

        GOTO verifica_passo;

    pos_93:
        !Posição 93

        !Carrega posição correspondente à familia selecionada
        IF GInput (PN_IN_Numero_Familia) = 1 THEN
            pPosição_Final_Buffer := pBuffer_Pos_93_Fam_1;
        ENDIF
        IF GInput (PN_IN_Numero_Familia) = 2 THEN
            pPosição_Final_Buffer := pBuffer_Pos_93_Fam_2;
        ENDIF
        IF GInput (PN_IN_Numero_Familia) = 3 THEN
            pPosição_Final_Buffer := pBuffer_Pos_93_Fam_3;
        ENDIF
        IF GInput (PN_IN_Numero_Familia) = 4 THEN
            pPosição_Final_Buffer := pBuffer_Pos_93_Fam_4;
        ENDIF

        GOTO verifica_passo;

    pos_94:
        !Posição 94

        !Carrega posição correspondente à familia selecionada
        IF GInput (PN_IN_Numero_Familia) = 1 THEN
            pPosição_Final_Buffer := pBuffer_Pos_94_Fam_1;
        ENDIF
        IF GInput (PN_IN_Numero_Familia) = 2 THEN
            pPosição_Final_Buffer := pBuffer_Pos_94_Fam_2;
        ENDIF
        IF GInput (PN_IN_Numero_Familia) = 3 THEN
            pPosição_Final_Buffer := pBuffer_Pos_94_Fam_3;
        ENDIF
        IF GInput (PN_IN_Numero_Familia) = 4 THEN
            pPosição_Final_Buffer := pBuffer_Pos_94_Fam_4;
        ENDIF

        GOTO verifica_passo;

    pos_95:
        !Posição 95

        !Carrega posição correspondente à familia selecionada
        IF GInput (PN_IN_Numero_Familia) = 1 THEN
            pPosição_Final_Buffer := pBuffer_Pos_95_Fam_1;
        ENDIF
        IF GInput (PN_IN_Numero_Familia) = 2 THEN
            pPosição_Final_Buffer := pBuffer_Pos_95_Fam_2;
        ENDIF
        IF GInput (PN_IN_Numero_Familia) = 3 THEN
            pPosição_Final_Buffer := pBuffer_Pos_95_Fam_3;
        ENDIF
        IF GInput (PN_IN_Numero_Familia) = 4 THEN
            pPosição_Final_Buffer := pBuffer_Pos_95_Fam_4;
        ENDIF

        GOTO verifica_passo;

    pos_96:
        !Posição 96

        !Carrega posição correspondente à familia selecionada
        IF GInput (PN_IN_Numero_Familia) = 1 THEN
            pPosição_Final_Buffer := pBuffer_Pos_96_Fam_1;
        ENDIF
        IF GInput (PN_IN_Numero_Familia) = 2 THEN
            pPosição_Final_Buffer := pBuffer_Pos_96_Fam_2;
        ENDIF
        IF GInput (PN_IN_Numero_Familia) = 3 THEN
            pPosição_Final_Buffer := pBuffer_Pos_96_Fam_3;
        ENDIF
        IF GInput (PN_IN_Numero_Familia) = 4 THEN
            pPosição_Final_Buffer := pBuffer_Pos_96_Fam_4;
        ENDIF

        GOTO verifica_passo;

    pos_97:
        !Posição 97

        !Carrega posição correspondente à familia selecionada
        IF GInput (PN_IN_Numero_Familia) = 1 THEN
            pPosição_Final_Buffer := pBuffer_Pos_97_Fam_1;
        ENDIF
        IF GInput (PN_IN_Numero_Familia) = 2 THEN
            pPosição_Final_Buffer := pBuffer_Pos_97_Fam_2;
        ENDIF
        IF GInput (PN_IN_Numero_Familia) = 3 THEN
            pPosição_Final_Buffer := pBuffer_Pos_97_Fam_3;
        ENDIF
        IF GInput (PN_IN_Numero_Familia) = 4 THEN
            pPosição_Final_Buffer := pBuffer_Pos_97_Fam_4;
        ENDIF

        GOTO verifica_passo;

    pos_98:
        !Posição 98

        !Carrega posição correspondente à familia selecionada
        IF GInput (PN_IN_Numero_Familia) = 1 THEN
            pPosição_Final_Buffer := pBuffer_Pos_98_Fam_1;
        ENDIF
        IF GInput (PN_IN_Numero_Familia) = 2 THEN
            pPosição_Final_Buffer := pBuffer_Pos_98_Fam_2;
        ENDIF
        IF GInput (PN_IN_Numero_Familia) = 3 THEN
            pPosição_Final_Buffer := pBuffer_Pos_98_Fam_3;
        ENDIF
        IF GInput (PN_IN_Numero_Familia) = 4 THEN
            pPosição_Final_Buffer := pBuffer_Pos_98_Fam_4;
        ENDIF

        GOTO verifica_passo;

    pos_99:
        !Posição 99

        !Carrega posição correspondente à familia selecionada
        IF GInput (PN_IN_Numero_Familia) = 1 THEN
            pPosição_Final_Buffer := pBuffer_Pos_99_Fam_1;
        ENDIF
        IF GInput (PN_IN_Numero_Familia) = 2 THEN
            pPosição_Final_Buffer := pBuffer_Pos_99_Fam_2;
        ENDIF
        IF GInput (PN_IN_Numero_Familia) = 3 THEN
            pPosição_Final_Buffer := pBuffer_Pos_99_Fam_3;
        ENDIF
        IF GInput (PN_IN_Numero_Familia) = 4 THEN
            pPosição_Final_Buffer := pBuffer_Pos_99_Fam_4;
        ENDIF

        GOTO verifica_passo;

    verifica_passo:
        !Verifica Produto
        IF GInput (PN_IN_Numero_Familia) = 3 GOTO ver_fam_3;
        IF GInput (PN_IN_Numero_Familia) = 4 GOTO ver_Fam_4;

        !Verifica se ciclo é de pega peça ou deposita peça no buffer
        IF GInput (PN_IN_Numero_Programa) = 3 GOTO deposita_fam_1_2;
        IF GInput (PN_IN_Numero_Programa) = 4 GOTO pega_fam_1_2;

    ver_fam_3:
        !Verifica se ciclo é de pega peça ou deposita peça no buffer
        IF GInput (PN_IN_Numero_Programa) = 3 GOTO deposita_fam_3;
        IF GInput (PN_IN_Numero_Programa) = 4 GOTO pega_fam_3;

    ver_fam_4:
        !Verifica se ciclo é de pega peça ou deposita peça no buffer
        IF GInput (PN_IN_Numero_Programa) = 3 GOTO deposita_fam_4;
        IF GInput (PN_IN_Numero_Programa) = 4 GOTO pega_fam_4;

!*********************************************************************************************************************************************
!  DEPOSITA PRODUTO NO BUFFER FAMILIAS 1 E 2
!*********************************************************************************************************************************************

    deposita_fam_1_2:
        !Ciclo para depositar peça no buffer

        !Ponto intermediario centro de massa
        AccSet nAcc_Mov_Geral, nRamp_Mov_Geral;
        IF (nPos_Buffer >= 13 AND nPos_Buffer <= 15) OR (nPos_Buffer >= 19 AND nPos_Buffer <= 21) OR (nPos_Buffer >= 25 AND nPos_Buffer <= 27) OR (nPos_Buffer >= 31 AND nPos_Buffer <=33) OR (nPos_Buffer >= 37 AND nPos_Buffer <= 39) OR (nPos_Buffer >= 43 AND nPos_Buffer <= 45) OR (nPos_Buffer >= 49 AND nPos_Buffer <= 51) OR (nPos_Buffer >= 55 AND nPos_Buffer <=57) OR (nPos_Buffer >= 61 AND nPos_Buffer <= 63) OR (nPos_Buffer >= 67 AND nPos_Buffer <= 69) OR (nPos_Buffer >= 73 AND nPos_Buffer <= 75) OR (nPos_Buffer >= 79 AND nPos_Buffer <= 81) OR (nPos_Buffer >= 85 AND nPos_Buffer <= 87) OR (nPos_Buffer >= 91 AND nPos_Buffer <= 93) OR (nPos_Buffer >= 97 AND nPos_Buffer <= 99) THEN
        pIntermedCentroMassa := pPosição_Final_Buffer;
	    jposIntermedCentroMassa := CalcJointT(pIntermedCentroMassa, tGarra \WObj:=wBuffer_Dir);
        jposIntermedCentroMassa.robax.rax_2 := jposRecolhidoEsteira.robax.rax_2;
        jposIntermedCentroMassa.robax.rax_3 := jposRecolhidoEsteira.robax.rax_3;
        jposIntermedCentroMassa.robax.rax_4 := jposRecolhidoEsteira.robax.rax_4;
        jposIntermedCentroMassa.robax.rax_5 := jposRecolhidoEsteira.robax.rax_5;


        MoveAbsJ jposIntermedCentroMassa, sMov_Geral_Com_Produto, z200, tGarra\WObj:=wBuffer_Dir;
        GOTO inpos_fam_1_2;
        ENDIF

        IF (nPos_Buffer >= 1 AND nPos_Buffer <= 9) THEN
        pIntermedCentroMassa := pPosição_Final_Buffer;
	    jposIntermedCentroMassa := CalcJointT(pIntermedCentroMassa, tGarra \WObj:=wBuffer_Front);
        jposIntermedCentroMassa.robax.rax_2 := jposRecolhidoEsteira.robax.rax_2;
        jposIntermedCentroMassa.robax.rax_3 := jposRecolhidoEsteira.robax.rax_3;
        jposIntermedCentroMassa.robax.rax_4 := jposRecolhidoEsteira.robax.rax_4;
        jposIntermedCentroMassa.robax.rax_5 := jposRecolhidoEsteira.robax.rax_5;

        MoveAbsJ jposIntermedCentroMassa, sMov_Geral_Com_Produto, z200, tGarra\WObj:=wBuffer_Front;
        GOTO inpos_fam_1_2;
        ELSE
        pIntermedCentroMassa := pPosição_Final_Buffer;
	    jposIntermedCentroMassa := CalcJointT(pIntermedCentroMassa, tGarra \WObj:=wBuffer_Esq);
        jposIntermedCentroMassa.robax.rax_2 := jposRecolhidoEsteira.robax.rax_2;
        jposIntermedCentroMassa.robax.rax_3 := jposRecolhidoEsteira.robax.rax_3;
        jposIntermedCentroMassa.robax.rax_4 := jposRecolhidoEsteira.robax.rax_4;
        jposIntermedCentroMassa.robax.rax_5 := jposRecolhidoEsteira.robax.rax_5;

        MoveAbsJ jposIntermedCentroMassa, sMov_Geral_Com_Produto, z200, tGarra\WObj:=wBuffer_Esq;
        ENDIF


inpos_fam_1_2:
        !Agora sim, vai para posição acima do local de deposita
        pMov_Pega_Depos_Buffer := pPosição_Final_Buffer;
        pMov_Pega_Depos_Buffer.trans := pMov_Pega_Depos_Buffer.trans + pOfst_Acima_Buffer;
        IF (nPos_Buffer >= 13 AND nPos_Buffer <= 15) OR (nPos_Buffer >= 19 AND nPos_Buffer <= 21) OR (nPos_Buffer >= 25 AND nPos_Buffer <= 27) OR (nPos_Buffer >= 31 AND nPos_Buffer <=33) OR (nPos_Buffer >= 37 AND nPos_Buffer <= 39) OR (nPos_Buffer >= 43 AND nPos_Buffer <= 45) OR (nPos_Buffer >= 49 AND nPos_Buffer <= 51) OR (nPos_Buffer >= 55 AND nPos_Buffer <=57) OR (nPos_Buffer >= 61 AND nPos_Buffer <= 63) OR (nPos_Buffer >= 67 AND nPos_Buffer <= 69) OR (nPos_Buffer >= 73 AND nPos_Buffer <= 75) OR (nPos_Buffer >= 79 AND nPos_Buffer <= 81) OR (nPos_Buffer >= 85 AND nPos_Buffer <= 87) OR (nPos_Buffer >= 91 AND nPos_Buffer <= 93) OR (nPos_Buffer >= 97 AND nPos_Buffer <= 99) THEN
        MoveL pMov_Pega_Depos_Buffer, sMov_Geral_Com_Produto, fine, tGarra \WObj:=wBuffer_Dir;
        GOTO verifica_fam_1_2;
        ENDIF
        IF (nPos_Buffer >= 1 AND nPos_Buffer <= 9) THEN
        MoveL pMov_Pega_Depos_Buffer, sMov_Geral_Com_Produto, fine, tGarra \WObj:=wBuffer_Front;
        GOTO verifica_fam_1_2;
        ELSE
        MoveL pMov_Pega_Depos_Buffer, sMov_Geral_Com_Produto, fine, tGarra \WObj:=wBuffer_Esq;
        ENDIF

    verifica_fam_1_2:
        !Verifica se já existe peça na posição selecionada
        IF DInput (DI_Pres_Peça_Berço_1) = 0 AND DInput (DI_Pres_Peça_Berço_2) = 1 GOTO a_berço;

        !Caso exista produto no berço selecionado
        TPWrite "Já existe um produto na posição "\num:= nPos_Buffer;
        SetDO PN_OUT_Produto_Existente, 1;
        Stop;
        GOTO inpos_fam_1_2;

    a_berço:
        SetDO PN_OUT_Produto_Existente, 0;

        !Ponto acima do berço
        pMov_Pega_Depos_Buffer := pPosição_Final_Buffer;
        pMov_Pega_Depos_Buffer.trans := pMov_Pega_Depos_Buffer.trans + pOfst_Acima_Berço_Buffer;
        IF (nPos_Buffer >= 13 AND nPos_Buffer <= 15) OR (nPos_Buffer >= 19 AND nPos_Buffer <= 21) OR (nPos_Buffer >= 25 AND nPos_Buffer <= 27) OR (nPos_Buffer >= 31 AND nPos_Buffer <=33) OR (nPos_Buffer >= 37 AND nPos_Buffer <= 39) OR (nPos_Buffer >= 43 AND nPos_Buffer <= 45) OR (nPos_Buffer >= 49 AND nPos_Buffer <= 51) OR (nPos_Buffer >= 55 AND nPos_Buffer <=57) OR (nPos_Buffer >= 61 AND nPos_Buffer <= 63) OR (nPos_Buffer >= 67 AND nPos_Buffer <= 69) OR (nPos_Buffer >= 73 AND nPos_Buffer <= 75) OR (nPos_Buffer >= 79 AND nPos_Buffer <= 81) OR (nPos_Buffer >= 85 AND nPos_Buffer <= 87) OR (nPos_Buffer >= 91 AND nPos_Buffer <= 93) OR (nPos_Buffer >= 97 AND nPos_Buffer <= 99) THEN
        MoveL pMov_Pega_Depos_Buffer, sMov_Aprox_Berço_Com_Produto, z50, tGarra \WObj:=wBuffer_Dir;
        GOTO p_aprox;
        ENDIF
        IF (nPos_Buffer >= 1 AND nPos_Buffer <= 9) THEN
        MoveL pMov_Pega_Depos_Buffer, sMov_Aprox_Berço_Com_Produto, z50, tGarra \WObj:=wBuffer_Front;
        GOTO p_aprox;
        ELSE
        MoveL pMov_Pega_Depos_Buffer, sMov_Aprox_Berço_Com_Produto, z50, tGarra \WObj:=wBuffer_Esq;
        ENDIF

    p_aprox:
        !Ponto de aproximação
        AccSet nAcc_Mov_Pega_Depos, nRamp_Mov_Pega_Depos;
        motionsup \On \TuneValue:= nSens_Colid_Aprox;
        pMov_Pega_Depos_Buffer := pPosição_Final_Buffer;
        pMov_Pega_Depos_Buffer.trans := pMov_Pega_Depos_Buffer.trans + pOfst_Aprox_Pega_Depos_Buffer;
        IF (nPos_Buffer >= 13 AND nPos_Buffer <= 15) OR (nPos_Buffer >= 19 AND nPos_Buffer <= 21) OR (nPos_Buffer >= 25 AND nPos_Buffer <= 27) OR (nPos_Buffer >= 31 AND nPos_Buffer <=33) OR (nPos_Buffer >= 37 AND nPos_Buffer <= 39) OR (nPos_Buffer >= 43 AND nPos_Buffer <= 45) OR (nPos_Buffer >= 49 AND nPos_Buffer <= 51) OR (nPos_Buffer >= 55 AND nPos_Buffer <=57) OR (nPos_Buffer >= 61 AND nPos_Buffer <= 63) OR (nPos_Buffer >= 67 AND nPos_Buffer <= 69) OR (nPos_Buffer >= 73 AND nPos_Buffer <= 75) OR (nPos_Buffer >= 79 AND nPos_Buffer <= 81) OR (nPos_Buffer >= 85 AND nPos_Buffer <= 87) OR (nPos_Buffer >= 91 AND nPos_Buffer <= 93) OR (nPos_Buffer >= 97 AND nPos_Buffer <= 99) THEN
        MoveL pMov_Pega_Depos_Buffer, SMov_Fina, z50, tGarra \WObj:=wBuffer_Dir;
        GOTO p_ant_ag_1_2;
        ENDIF
        IF (nPos_Buffer >= 1 AND nPos_Buffer <= 9) THEN
        MoveL pMov_Pega_Depos_Buffer, SMov_Fina, z50, tGarra \WObj:=wBuffer_Front;
        GOTO p_ant_ag_1_2;
        ELSE
        MoveL pMov_Pega_Depos_Buffer, SMov_Fina, z50, tGarra \WObj:=wBuffer_Esq;
        ENDIF

    p_ant_ag_1_2:
        pMov_Pega_Depos_Buffer := pPosição_Final_Buffer;
        pMov_Pega_Depos_Buffer.trans := pMov_Pega_Depos_Buffer.trans + pOfst_Aprox_Final_Depos;
        IF (nPos_Buffer >= 13 AND nPos_Buffer <= 15) OR (nPos_Buffer >= 19 AND nPos_Buffer <= 21) OR (nPos_Buffer >= 25 AND nPos_Buffer <= 27) OR (nPos_Buffer >= 31 AND nPos_Buffer <=33) OR (nPos_Buffer >= 37 AND nPos_Buffer <= 39) OR (nPos_Buffer >= 43 AND nPos_Buffer <= 45) OR (nPos_Buffer >= 49 AND nPos_Buffer <= 51) OR (nPos_Buffer >= 55 AND nPos_Buffer <=57) OR (nPos_Buffer >= 61 AND nPos_Buffer <= 63) OR (nPos_Buffer >= 67 AND nPos_Buffer <= 69) OR (nPos_Buffer >= 73 AND nPos_Buffer <= 75) OR (nPos_Buffer >= 79 AND nPos_Buffer <= 81) OR (nPos_Buffer >= 85 AND nPos_Buffer <= 87) OR (nPos_Buffer >= 91 AND nPos_Buffer <= 93) OR (nPos_Buffer >= 97 AND nPos_Buffer <= 99) THEN
        MoveL pMov_Pega_Depos_Buffer, SMov_SuperFina, z1, tGarra\WObj:=wBuffer_Dir;
        GOTO  p_depos;
        ENDIF
        IF (nPos_Buffer >= 1 AND nPos_Buffer <= 9) THEN
        MoveL pMov_Pega_Depos_Buffer, SMov_SuperFina, z1, tGarra \WObj:=wBuffer_Front;
        GOTO  p_depos;
        ELSE
        MoveL pMov_Pega_Depos_Buffer, SMov_SuperFina, z1, tGarra \WObj:=wBuffer_Esq;
        ENDIF

    p_depos:
        !Destrava o produto
        GARRA_DestravarProduto;

        !Ponto final para depositar
        pMov_Pega_Depos_Buffer := pPosição_Final_Buffer;
        IF (nPos_Buffer >= 13 AND nPos_Buffer <= 15) OR (nPos_Buffer >= 19 AND nPos_Buffer <= 21) OR (nPos_Buffer >= 25 AND nPos_Buffer <= 27) OR (nPos_Buffer >= 31 AND nPos_Buffer <=33) OR (nPos_Buffer >= 37 AND nPos_Buffer <= 39) OR (nPos_Buffer >= 43 AND nPos_Buffer <= 45) OR (nPos_Buffer >= 49 AND nPos_Buffer <= 51) OR (nPos_Buffer >= 55 AND nPos_Buffer <=57) OR (nPos_Buffer >= 61 AND nPos_Buffer <= 63) OR (nPos_Buffer >= 67 AND nPos_Buffer <= 69) OR (nPos_Buffer >= 73 AND nPos_Buffer <= 75) OR (nPos_Buffer >= 79 AND nPos_Buffer <= 81) OR (nPos_Buffer >= 85 AND nPos_Buffer <= 87) OR (nPos_Buffer >= 91 AND nPos_Buffer <= 93) OR (nPos_Buffer >= 97 AND nPos_Buffer <= 99) THEN
        MoveL pMov_Pega_Depos_Buffer, SMov_SuperFina, fine, tGarra\WObj:=wBuffer_Dir;
        GOTO a_garra;
        ENDIF
        IF (nPos_Buffer >= 1 AND nPos_Buffer <= 9) THEN
        MoveL pMov_Pega_Depos_Buffer, SMov_SuperFina, fine, tGarra \WObj:=wBuffer_Front;
        GOTO a_garra;
        ELSE
        MoveL pMov_Pega_Depos_Buffer, SMov_SuperFina, fine, tGarra \WObj:=wBuffer_Esq;
        ENDIF


      a_garra:
        !Deposita Produto
        GARRA_AbrirGarra;

        GripLoad load0;

        !Movimento de Recuo
        pMov_Pega_Depos_Buffer := pPosição_Final_Buffer;
        pMov_Pega_Depos_Buffer.trans := pMov_Pega_Depos_Buffer.trans + pOfst_Acima_Berço_Buffer;
        IF (nPos_Buffer >= 13 AND nPos_Buffer <= 15) OR (nPos_Buffer >= 19 AND nPos_Buffer <= 21) OR (nPos_Buffer >= 25 AND nPos_Buffer <= 27) OR (nPos_Buffer >= 31 AND nPos_Buffer <=33) OR (nPos_Buffer >= 37 AND nPos_Buffer <= 39) OR (nPos_Buffer >= 43 AND nPos_Buffer <= 45) OR (nPos_Buffer >= 49 AND nPos_Buffer <= 51) OR (nPos_Buffer >= 55 AND nPos_Buffer <=57) OR (nPos_Buffer >= 61 AND nPos_Buffer <= 63) OR (nPos_Buffer >= 67 AND nPos_Buffer <= 69) OR (nPos_Buffer >= 73 AND nPos_Buffer <= 75) OR (nPos_Buffer >= 79 AND nPos_Buffer <= 81) OR (nPos_Buffer >= 85 AND nPos_Buffer <= 87) OR (nPos_Buffer >= 91 AND nPos_Buffer <= 93) OR (nPos_Buffer >= 97 AND nPos_Buffer <= 99) THEN
        MoveL pMov_Pega_Depos_Buffer, sMov_Aprox_Berço_Sem_Produto, z50, tGarra \WObj:=wBuffer_Dir;
        GOTO ad_buffer;
        ENDIF
        IF (nPos_Buffer >= 1 AND nPos_Buffer <= 9) THEN
        MoveL pMov_Pega_Depos_Buffer, sMov_Aprox_Berço_Sem_Produto, z50, tGarra \WObj:=wBuffer_Front;
        GOTO ad_buffer;
        ELSE
        MoveL pMov_Pega_Depos_Buffer, sMov_Aprox_Berço_Sem_Produto, z50, tGarra \WObj:=wBuffer_Esq;
        ENDIF

    ad_buffer:
        AccSet nAcc_Mov_Geral, nRamp_Mov_Geral;
        motionsup \On \TuneValue:= nSens_Colid_Mov_Geral;
        pMov_Pega_Depos_Buffer := pPosição_Final_Buffer;
        pMov_Pega_Depos_Buffer.trans := pMov_Pega_Depos_Buffer.trans + pOfst_Acima_Buffer_Sem_Produto;
        IF (nPos_Buffer >= 13 AND nPos_Buffer <= 15) OR (nPos_Buffer >= 19 AND nPos_Buffer <= 21) OR (nPos_Buffer >= 25 AND nPos_Buffer <= 27) OR (nPos_Buffer >= 31 AND nPos_Buffer <=33) OR (nPos_Buffer >= 37 AND nPos_Buffer <= 39) OR (nPos_Buffer >= 43 AND nPos_Buffer <= 45) OR (nPos_Buffer >= 49 AND nPos_Buffer <= 51) OR (nPos_Buffer >= 55 AND nPos_Buffer <=57) OR (nPos_Buffer >= 61 AND nPos_Buffer <= 63) OR (nPos_Buffer >= 67 AND nPos_Buffer <= 69) OR (nPos_Buffer >= 73 AND nPos_Buffer <= 75) OR (nPos_Buffer >= 79 AND nPos_Buffer <= 81) OR (nPos_Buffer >= 85 AND nPos_Buffer <= 87) OR (nPos_Buffer >= 91 AND nPos_Buffer <= 93) OR (nPos_Buffer >= 97 AND nPos_Buffer <= 99) THEN
        MoveL pMov_Pega_Depos_Buffer, sMov_Geral_Sem_Produto, z200, tGarra \WObj:=wBuffer_Dir;
        GOTO inposf_fam_1_2;
        ENDIF
        IF (nPos_Buffer >= 1 AND nPos_Buffer <= 9) THEN
        MoveL pMov_Pega_Depos_Buffer, sMov_Geral_Sem_Produto, z200, tGarra \WObj:=wBuffer_Front;
        GOTO inposf_fam_1_2;
        ELSE
        MoveL pMov_Pega_Depos_Buffer, sMov_Geral_Sem_Produto, z200, tGarra \WObj:=wBuffer_Esq;
        ENDIF
        GOTO inposf_fam_1_2;

    inposf_fam_1_2:
        IF (nPos_Buffer >= 13 AND nPos_Buffer <= 15) OR (nPos_Buffer >= 19 AND nPos_Buffer <= 21) OR (nPos_Buffer >= 25 AND nPos_Buffer <= 27) OR (nPos_Buffer >= 31 AND nPos_Buffer <=33) OR (nPos_Buffer >= 37 AND nPos_Buffer <= 39) OR (nPos_Buffer >= 43 AND nPos_Buffer <= 45) OR (nPos_Buffer >= 49 AND nPos_Buffer <= 51) OR (nPos_Buffer >= 55 AND nPos_Buffer <=57) OR (nPos_Buffer >= 61 AND nPos_Buffer <= 63) OR (nPos_Buffer >= 67 AND nPos_Buffer <= 69) OR (nPos_Buffer >= 73 AND nPos_Buffer <= 75) OR (nPos_Buffer >= 79 AND nPos_Buffer <= 81) OR (nPos_Buffer >= 85 AND nPos_Buffer <= 87) OR (nPos_Buffer >= 91 AND nPos_Buffer <= 93) OR (nPos_Buffer >= 97 AND nPos_Buffer <= 99) THEN
        MoveAbsJ jposIntermedCentroMassa, sMov_Geral_Sem_Produto, z200, tGarra\WObj:=wBuffer_Dir;
        GOTO final;
        ENDIF
        IF (nPos_Buffer >= 1 AND nPos_Buffer <= 9) THEN
        MoveAbsJ jposIntermedCentroMassa, sMov_Geral_Sem_Produto, z200, tGarra\WObj:=wBuffer_Front;
        GOTO final;
        ELSE
        MoveAbsJ jposIntermedCentroMassa, sMov_Geral_Sem_Produto, z200, tGarra\WObj:=wBuffer_Esq;
        ENDIF
        GOTO final;

!*********************************************************************************************************************************************
!  PEGA PRODUTO NO BUFFER FAMILIAS 1 E 2
!*********************************************************************************************************************************************
    pega_fam_1_2:
        !Ciclo para pegar peça no buffer

        GARRA_VerificarGarraVazia;
        !Abre Garra
        GARRA_DestravarProduto;
        GARRA_AbrirGarra;

        !Vai para posição intermediária no centro de massa
        AccSet nAcc_Mov_Geral, nRamp_Mov_Geral;

        IF (nPos_Buffer >= 13 AND nPos_Buffer <= 15) OR (nPos_Buffer >= 19 AND nPos_Buffer <= 21) OR (nPos_Buffer >= 25 AND nPos_Buffer <= 27) OR (nPos_Buffer >= 31 AND nPos_Buffer <=33) OR (nPos_Buffer >= 37 AND nPos_Buffer <= 39) OR (nPos_Buffer >= 43 AND nPos_Buffer <= 45) OR (nPos_Buffer >= 49 AND nPos_Buffer <= 51) OR (nPos_Buffer >= 55 AND nPos_Buffer <=57) OR (nPos_Buffer >= 61 AND nPos_Buffer <= 63) OR (nPos_Buffer >= 67 AND nPos_Buffer <= 69) OR (nPos_Buffer >= 73 AND nPos_Buffer <= 75) OR (nPos_Buffer >= 79 AND nPos_Buffer <= 81) OR (nPos_Buffer >= 85 AND nPos_Buffer <= 87) OR (nPos_Buffer >= 91 AND nPos_Buffer <= 93) OR (nPos_Buffer >= 97 AND nPos_Buffer <= 99) THEN
        pIntermedCentroMassa := pPosição_Final_Buffer;
	    jposIntermedCentroMassa := CalcJointT(pIntermedCentroMassa, tGarra \WObj:=wBuffer_Dir);
        jposIntermedCentroMassa.robax.rax_2 := jposRecolhidoEsteira.robax.rax_2;
        jposIntermedCentroMassa.robax.rax_3 := jposRecolhidoEsteira.robax.rax_3;
        jposIntermedCentroMassa.robax.rax_4 := jposRecolhidoEsteira.robax.rax_4;
        jposIntermedCentroMassa.robax.rax_5 := jposRecolhidoEsteira.robax.rax_5;

        MoveAbsJ jposIntermedCentroMassa, sMov_Geral_Sem_Produto, z200, tGarra\WObj:=wBuffer_Dir;
        GOTO inpegapos_fam_1_2;
        ENDIF

        IF (nPos_Buffer >= 1 AND nPos_Buffer <= 9) THEN
        pIntermedCentroMassa := pPosição_Final_Buffer;
	    jposIntermedCentroMassa := CalcJointT(pIntermedCentroMassa, tGarra \WObj:=wBuffer_Front);
        jposIntermedCentroMassa.robax.rax_2 := jposRecolhidoEsteira.robax.rax_2;
        jposIntermedCentroMassa.robax.rax_3 := jposRecolhidoEsteira.robax.rax_3;
        jposIntermedCentroMassa.robax.rax_4 := jposRecolhidoEsteira.robax.rax_4;
        jposIntermedCentroMassa.robax.rax_5 := jposRecolhidoEsteira.robax.rax_5;

        MoveAbsJ jposIntermedCentroMassa, sMov_Geral_Sem_Produto, z200, tGarra\WObj:=wBuffer_Front;
        GOTO inpegapos_fam_1_2;
        ELSE
        pIntermedCentroMassa := pPosição_Final_Buffer;
	    jposIntermedCentroMassa := CalcJointT(pIntermedCentroMassa, tGarra \WObj:=wBuffer_Esq);
        jposIntermedCentroMassa.robax.rax_2 := jposRecolhidoEsteira.robax.rax_2;
        jposIntermedCentroMassa.robax.rax_3 := jposRecolhidoEsteira.robax.rax_3;
        jposIntermedCentroMassa.robax.rax_4 := jposRecolhidoEsteira.robax.rax_4;
        jposIntermedCentroMassa.robax.rax_5 := jposRecolhidoEsteira.robax.rax_5;

        MoveAbsJ jposIntermedCentroMassa, sMov_Geral_Sem_Produto, z200, tGarra\WObj:=wBuffer_Esq;
        ENDIF

    inpegapos_fam_1_2:
        !Ponto acima da posição
        AccSet nAcc_Mov_Geral, nRamp_Mov_Geral;
        pMov_Pega_Depos_Buffer := pPosição_Final_Buffer;
        pMov_Pega_Depos_Buffer.trans := pMov_Pega_Depos_Buffer.trans + pOfst_Acima_Buffer_Sem_Produto;
        IF (nPos_Buffer >= 13 AND nPos_Buffer <= 15) OR (nPos_Buffer >= 19 AND nPos_Buffer <= 21) OR (nPos_Buffer >= 25 AND nPos_Buffer <= 27) OR (nPos_Buffer >= 31 AND nPos_Buffer <=33) OR (nPos_Buffer >= 37 AND nPos_Buffer <= 39) OR (nPos_Buffer >= 43 AND nPos_Buffer <= 45) OR (nPos_Buffer >= 49 AND nPos_Buffer <= 51) OR (nPos_Buffer >= 55 AND nPos_Buffer <=57) OR (nPos_Buffer >= 61 AND nPos_Buffer <= 63) OR (nPos_Buffer >= 67 AND nPos_Buffer <= 69) OR (nPos_Buffer >= 73 AND nPos_Buffer <= 75) OR (nPos_Buffer >= 79 AND nPos_Buffer <= 81) OR (nPos_Buffer >= 85 AND nPos_Buffer <= 87) OR (nPos_Buffer >= 91 AND nPos_Buffer <= 93) OR (nPos_Buffer >= 97 AND nPos_Buffer <= 99) THEN
        MoveL pMov_Pega_Depos_Buffer, sMov_Geral_Sem_Produto, fine, tGarra \WObj:=wBuffer_Dir;
        GOTO  ap_berço;
        ENDIF
        IF (nPos_Buffer >= 1 AND nPos_Buffer <= 9) THEN
        MoveL pMov_Pega_Depos_Buffer, sMov_Geral_Sem_Produto, fine, tGarra \WObj:=wBuffer_Front;
        GOTO  ap_berço;
        ELSE
        MoveL pMov_Pega_Depos_Buffer, sMov_Geral_Sem_Produto, fine, tGarra \WObj:=wBuffer_Esq;
        ENDIF

     ap_berço:
        !Ponto acima do berço
        pMov_Pega_Depos_Buffer := pPosição_Final_Buffer;
        pMov_Pega_Depos_Buffer.trans := pMov_Pega_Depos_Buffer.trans + pOfst_Acima_Berço_Buffer;
        IF (nPos_Buffer >= 13 AND nPos_Buffer <= 15) OR (nPos_Buffer >= 19 AND nPos_Buffer <= 21) OR (nPos_Buffer >= 25 AND nPos_Buffer <= 27) OR (nPos_Buffer >= 31 AND nPos_Buffer <=33) OR (nPos_Buffer >= 37 AND nPos_Buffer <= 39) OR (nPos_Buffer >= 43 AND nPos_Buffer <= 45) OR (nPos_Buffer >= 49 AND nPos_Buffer <= 51) OR (nPos_Buffer >= 55 AND nPos_Buffer <=57) OR (nPos_Buffer >= 61 AND nPos_Buffer <= 63) OR (nPos_Buffer >= 67 AND nPos_Buffer <= 69) OR (nPos_Buffer >= 73 AND nPos_Buffer <= 75) OR (nPos_Buffer >= 79 AND nPos_Buffer <= 81) OR (nPos_Buffer >= 85 AND nPos_Buffer <= 87) OR (nPos_Buffer >= 91 AND nPos_Buffer <= 93) OR (nPos_Buffer >= 97 AND nPos_Buffer <= 99) THEN
        MoveL pMov_Pega_Depos_Buffer, sMov_Aprox_Berço_Sem_Produto, z100, tGarra \WObj:=wBuffer_Dir;
        GOTO  pp_aprox;
        ENDIF
        IF (nPos_Buffer >= 1 AND nPos_Buffer <= 9) THEN
        MoveL pMov_Pega_Depos_Buffer, sMov_Aprox_Berço_Sem_Produto, z100, tGarra \WObj:=wBuffer_Front;
        GOTO  pp_aprox;
        ELSE
        MoveL pMov_Pega_Depos_Buffer, sMov_Aprox_Berço_Sem_Produto, z100, tGarra \WObj:=wBuffer_Esq;
        ENDIF

    pp_aprox:
        !Ponto de aproximação
        motionsup \On \TuneValue:= nSens_Colid_Aprox;
        pMov_Pega_Depos_Buffer := pPosição_Final_Buffer;
        pMov_Pega_Depos_Buffer.trans := pMov_Pega_Depos_Buffer.trans + pOfst_Aprox_Pega_Depos_Buffer;
        IF (nPos_Buffer >= 13 AND nPos_Buffer <= 15) OR (nPos_Buffer >= 19 AND nPos_Buffer <= 21) OR (nPos_Buffer >= 25 AND nPos_Buffer <= 27) OR (nPos_Buffer >= 31 AND nPos_Buffer <=33) OR (nPos_Buffer >= 37 AND nPos_Buffer <= 39) OR (nPos_Buffer >= 43 AND nPos_Buffer <= 45) OR (nPos_Buffer >= 49 AND nPos_Buffer <= 51) OR (nPos_Buffer >= 55 AND nPos_Buffer <=57) OR (nPos_Buffer >= 61 AND nPos_Buffer <= 63) OR (nPos_Buffer >= 67 AND nPos_Buffer <= 69) OR (nPos_Buffer >= 73 AND nPos_Buffer <= 75) OR (nPos_Buffer >= 79 AND nPos_Buffer <= 81) OR (nPos_Buffer >= 85 AND nPos_Buffer <= 87) OR (nPos_Buffer >= 91 AND nPos_Buffer <= 93) OR (nPos_Buffer >= 97 AND nPos_Buffer <= 99) THEN
        MoveL pMov_Pega_Depos_Buffer, SMov_Fina, z50, tGarra \WObj:=wBuffer_Dir;
        GOTO  p_peça;
        ENDIF
        IF (nPos_Buffer >= 1 AND nPos_Buffer <= 9) THEN
        MoveL pMov_Pega_Depos_Buffer, SMov_Fina, z50, tGarra \WObj:=wBuffer_Front;
        GOTO  p_peça;
        ELSE
        MoveL pMov_Pega_Depos_Buffer, SMov_Fina, z50, tGarra \WObj:=wBuffer_Esq;
        ENDIF

    p_peça:
        !Ponto de pega
        pMov_Pega_Depos_Buffer := pPosição_Final_Buffer;
        IF (nPos_Buffer >= 13 AND nPos_Buffer <= 15) OR (nPos_Buffer >= 19 AND nPos_Buffer <= 21) OR (nPos_Buffer >= 25 AND nPos_Buffer <= 27) OR (nPos_Buffer >= 31 AND nPos_Buffer <=33) OR (nPos_Buffer >= 37 AND nPos_Buffer <= 39) OR (nPos_Buffer >= 43 AND nPos_Buffer <= 45) OR (nPos_Buffer >= 49 AND nPos_Buffer <= 51) OR (nPos_Buffer >= 55 AND nPos_Buffer <=57) OR (nPos_Buffer >= 61 AND nPos_Buffer <= 63) OR (nPos_Buffer >= 67 AND nPos_Buffer <= 69) OR (nPos_Buffer >= 73 AND nPos_Buffer <= 75) OR (nPos_Buffer >= 79 AND nPos_Buffer <= 81) OR (nPos_Buffer >= 85 AND nPos_Buffer <= 87) OR (nPos_Buffer >= 91 AND nPos_Buffer <= 93) OR (nPos_Buffer >= 97 AND nPos_Buffer <= 99) THEN
        MoveL pMov_Pega_Depos_Buffer, SMov_SuperFina, fine, tGarra \WObj:=wBuffer_Dir;
        GOTO f_garra;
        ENDIF
        IF (nPos_Buffer >= 1 AND nPos_Buffer <= 9) THEN
        MoveL pMov_Pega_Depos_Buffer, SMov_SuperFina, fine, tGarra \WObj:=wBuffer_Front;
        GOTO f_garra;
        ELSE
        MoveL pMov_Pega_Depos_Buffer, SMov_SuperFina, fine, tGarra \WObj:=wBuffer_Esq;
        ENDIF

    f_garra:
        !Pega Produto
        GARRA_FecharGarra;

        TEST nNum_Fam
          CASE 1:
            GripLoad lFamilia_1;
          CASE 2:
            GripLoad lFamilia_2;
          DEFAULT:
            EXIT;
        ENDTEST

        !Movimento de Recuo
        AccSet nAcc_Mov_Pega_Depos, nRamp_Mov_Pega_Depos;

        pMov_Pega_Depos_Buffer := pPosição_Final_Buffer;
        pMov_Pega_Depos_Buffer.trans := pMov_Pega_Depos_Buffer.trans + pOfst_Aprox_Inicial_Pega;
        IF (nPos_Buffer >= 13 AND nPos_Buffer <= 15) OR (nPos_Buffer >= 19 AND nPos_Buffer <= 21) OR (nPos_Buffer >= 25 AND nPos_Buffer <= 27) OR (nPos_Buffer >= 31 AND nPos_Buffer <=33) OR (nPos_Buffer >= 37 AND nPos_Buffer <= 39) OR (nPos_Buffer >= 43 AND nPos_Buffer <= 45) OR (nPos_Buffer >= 49 AND nPos_Buffer <= 51) OR (nPos_Buffer >= 55 AND nPos_Buffer <=57) OR (nPos_Buffer >= 61 AND nPos_Buffer <= 63) OR (nPos_Buffer >= 67 AND nPos_Buffer <= 69) OR (nPos_Buffer >= 73 AND nPos_Buffer <= 75) OR (nPos_Buffer >= 79 AND nPos_Buffer <= 81) OR (nPos_Buffer >= 85 AND nPos_Buffer <= 87) OR (nPos_Buffer >= 91 AND nPos_Buffer <= 93) OR (nPos_Buffer >= 97 AND nPos_Buffer <= 99) THEN
        MoveL pMov_Pega_Depos_Buffer, SMov_SuperFina, z1, tGarra \WObj:=wBuffer_Dir;
        GOTO  tp_ac_1_2;
        ENDIF
        IF (nPos_Buffer >= 1 AND nPos_Buffer <= 9) THEN
        MoveL pMov_Pega_Depos_Buffer, SMov_SuperFina, z1, tGarra \WObj:=wBuffer_Front;
        GOTO  tp_ac_1_2;
        ELSE
        MoveL pMov_Pega_Depos_Buffer, SMov_SuperFina, z1, tGarra \WObj:=wBuffer_Esq;
        ENDIF

    tp_ac_1_2:
        !Trava o produto
        GARRA_TravarProduto;

        pMov_Pega_Depos_Buffer := pPosição_Final_Buffer;
        pMov_Pega_Depos_Buffer.trans := pMov_Pega_Depos_Buffer.trans + pOfst_Aprox_Pega_Depos_Buffer;
        IF (nPos_Buffer >= 13 AND nPos_Buffer <= 15) OR (nPos_Buffer >= 19 AND nPos_Buffer <= 21) OR (nPos_Buffer >= 25 AND nPos_Buffer <= 27) OR (nPos_Buffer >= 31 AND nPos_Buffer <=33) OR (nPos_Buffer >= 37 AND nPos_Buffer <= 39) OR (nPos_Buffer >= 43 AND nPos_Buffer <= 45) OR (nPos_Buffer >= 49 AND nPos_Buffer <= 51) OR (nPos_Buffer >= 55 AND nPos_Buffer <=57) OR (nPos_Buffer >= 61 AND nPos_Buffer <= 63) OR (nPos_Buffer >= 67 AND nPos_Buffer <= 69) OR (nPos_Buffer >= 73 AND nPos_Buffer <= 75) OR (nPos_Buffer >= 79 AND nPos_Buffer <= 81) OR (nPos_Buffer >= 85 AND nPos_Buffer <= 87) OR (nPos_Buffer >= 91 AND nPos_Buffer <= 93) OR (nPos_Buffer >= 97 AND nPos_Buffer <= 99) THEN
        MoveL pMov_Pega_Depos_Buffer, SMov_Levanta_Com_Produto, z50, tGarra \WObj:=wBuffer_Dir;
        GOTO  tp_buffer;
        ENDIF
        IF (nPos_Buffer >= 1 AND nPos_Buffer <= 9) THEN
        MoveL pMov_Pega_Depos_Buffer, SMov_Levanta_Com_Produto, z50, tGarra \WObj:=wBuffer_Front;
        GOTO  tp_buffer;
        ELSE
        MoveL pMov_Pega_Depos_Buffer, SMov_Levanta_Com_Produto, z50, tGarra \WObj:=wBuffer_Esq;
        ENDIF

    tp_buffer:
        pMov_Pega_Depos_Buffer := pPosição_Final_Buffer;
        pMov_Pega_Depos_Buffer.trans := pMov_Pega_Depos_Buffer.trans + pOfst_Acima_Berço_Buffer;
        IF (nPos_Buffer >= 13 AND nPos_Buffer <= 15) OR (nPos_Buffer >= 19 AND nPos_Buffer <= 21) OR (nPos_Buffer >= 25 AND nPos_Buffer <= 27) OR (nPos_Buffer >= 31 AND nPos_Buffer <=33) OR (nPos_Buffer >= 37 AND nPos_Buffer <= 39) OR (nPos_Buffer >= 43 AND nPos_Buffer <= 45) OR (nPos_Buffer >= 49 AND nPos_Buffer <= 51) OR (nPos_Buffer >= 55 AND nPos_Buffer <=57) OR (nPos_Buffer >= 61 AND nPos_Buffer <= 63) OR (nPos_Buffer >= 67 AND nPos_Buffer <= 69) OR (nPos_Buffer >= 73 AND nPos_Buffer <= 75) OR (nPos_Buffer >= 79 AND nPos_Buffer <= 81) OR (nPos_Buffer >= 85 AND nPos_Buffer <= 87) OR (nPos_Buffer >= 91 AND nPos_Buffer <= 93) OR (nPos_Buffer >= 97 AND nPos_Buffer <= 99) THEN
        MoveL pMov_Pega_Depos_Buffer, SMov_Levanta_Com_Produto, z80, tGarra\WObj:=wBuffer_Dir;
        GOTO  ap_buffer;
        ENDIF
        IF (nPos_Buffer >= 1 AND nPos_Buffer <= 9) THEN
        MoveL pMov_Pega_Depos_Buffer, SMov_Levanta_Com_Produto, z80, tGarra \WObj:=wBuffer_Front;
        GOTO  ap_buffer;
        ELSE
        MoveL pMov_Pega_Depos_Buffer, SMov_Levanta_Com_Produto, z80, tGarra \WObj:=wBuffer_Esq;
        ENDIF

    ap_buffer:
        AccSet nAcc_Mov_Geral, nRamp_Mov_Geral;
        motionsup \On \TuneValue:= nSens_Colid_Mov_Geral;
        pMov_Pega_Depos_Buffer := pPosição_Final_Buffer;
        pMov_Pega_Depos_Buffer.trans := pMov_Pega_Depos_Buffer.trans + pOfst_Acima_Buffer;
        IF (nPos_Buffer >= 13 AND nPos_Buffer <= 15) OR (nPos_Buffer >= 19 AND nPos_Buffer <= 21) OR (nPos_Buffer >= 25 AND nPos_Buffer <= 27) OR (nPos_Buffer >= 31 AND nPos_Buffer <=33) OR (nPos_Buffer >= 37 AND nPos_Buffer <= 39) OR (nPos_Buffer >= 43 AND nPos_Buffer <= 45) OR (nPos_Buffer >= 49 AND nPos_Buffer <= 51) OR (nPos_Buffer >= 55 AND nPos_Buffer <=57) OR (nPos_Buffer >= 61 AND nPos_Buffer <= 63) OR (nPos_Buffer >= 67 AND nPos_Buffer <= 69) OR (nPos_Buffer >= 73 AND nPos_Buffer <= 75) OR (nPos_Buffer >= 79 AND nPos_Buffer <= 81) OR (nPos_Buffer >= 85 AND nPos_Buffer <= 87) OR (nPos_Buffer >= 91 AND nPos_Buffer <= 93) OR (nPos_Buffer >= 97 AND nPos_Buffer <= 99) THEN
        MoveL pMov_Pega_Depos_Buffer, sMov_Aprox_Berço_Com_Produto, z100, tGarra \WObj:=wBuffer_Dir;
        GOTO  inpegaposf_fam_1_2;
        ENDIF
        IF (nPos_Buffer >= 1 AND nPos_Buffer <= 9) THEN
        MoveL pMov_Pega_Depos_Buffer, sMov_Aprox_Berço_Com_Produto, z100, tGarra \WObj:=wBuffer_Front;
        GOTO  inpegaposf_fam_1_2;
        ELSE
        MoveL pMov_Pega_Depos_Buffer, sMov_Aprox_Berço_Com_Produto, z100, tGarra \WObj:=wBuffer_Esq;
        ENDIF
        GOTO inpegaposf_fam_1_2;

    inpegaposf_fam_1_2:
        IF (nPos_Buffer >= 13 AND nPos_Buffer <= 15) OR (nPos_Buffer >= 19 AND nPos_Buffer <= 21) OR (nPos_Buffer >= 25 AND nPos_Buffer <= 27) OR (nPos_Buffer >= 31 AND nPos_Buffer <=33) OR (nPos_Buffer >= 37 AND nPos_Buffer <= 39) OR (nPos_Buffer >= 43 AND nPos_Buffer <= 45) OR (nPos_Buffer >= 49 AND nPos_Buffer <= 51) OR (nPos_Buffer >= 55 AND nPos_Buffer <=57) OR (nPos_Buffer >= 61 AND nPos_Buffer <= 63) OR (nPos_Buffer >= 67 AND nPos_Buffer <= 69) OR (nPos_Buffer >= 73 AND nPos_Buffer <= 75) OR (nPos_Buffer >= 79 AND nPos_Buffer <= 81) OR (nPos_Buffer >= 85 AND nPos_Buffer <= 87) OR (nPos_Buffer >= 91 AND nPos_Buffer <= 93) OR (nPos_Buffer >= 97 AND nPos_Buffer <= 99) THEN
        MoveAbsJ jposIntermedCentroMassa, sMov_Geral_Com_Produto, z200, tGarra\WObj:=wBuffer_Dir;
        GOTO  final;
        ENDIF
        IF (nPos_Buffer >= 1 AND nPos_Buffer <= 9) THEN
        MoveAbsJ jposIntermedCentroMassa, sMov_Geral_Com_Produto, z200, tGarra\WObj:=wBuffer_Front;
        GOTO  final;
        ELSE
        MoveAbsJ jposIntermedCentroMassa, sMov_Geral_Com_Produto, z200, tGarra\WObj:=wBuffer_Esq;
        ENDIF
        GOTO final;

!*********************************************************************************************************************************************
!  DEPOSITA PRODUTO NO BUFFER FAMILIA 3
!*********************************************************************************************************************************************

    deposita_fam_3:
        !Ciclo para depositar peça no buffer

        !Ponto intermediario centro de massa
        AccSet nAcc_Mov_Geral, nRamp_Mov_Geral;
        IF (nPos_Buffer >= 13 AND nPos_Buffer <= 15) OR (nPos_Buffer >= 19 AND nPos_Buffer <= 21) OR (nPos_Buffer >= 25 AND nPos_Buffer <= 27) OR (nPos_Buffer >= 31 AND nPos_Buffer <=33) OR (nPos_Buffer >= 37 AND nPos_Buffer <= 39) OR (nPos_Buffer >= 43 AND nPos_Buffer <= 45) OR (nPos_Buffer >= 49 AND nPos_Buffer <= 51) OR (nPos_Buffer >= 55 AND nPos_Buffer <=57) OR (nPos_Buffer >= 61 AND nPos_Buffer <= 63) OR (nPos_Buffer >= 67 AND nPos_Buffer <= 69) OR (nPos_Buffer >= 73 AND nPos_Buffer <= 75) OR (nPos_Buffer >= 79 AND nPos_Buffer <= 81) OR (nPos_Buffer >= 85 AND nPos_Buffer <= 87) OR (nPos_Buffer >= 91 AND nPos_Buffer <= 93) OR (nPos_Buffer >= 97 AND nPos_Buffer <= 99) THEN
        pIntermedCentroMassa := pPosição_Final_Buffer;
	    jposIntermedCentroMassa := CalcJointT(pIntermedCentroMassa, tGarra \WObj:=wBuffer_Dir);
        jposIntermedCentroMassa.robax.rax_2 := jposRecolhidoEsteira.robax.rax_2;
        jposIntermedCentroMassa.robax.rax_3 := jposRecolhidoEsteira.robax.rax_3;
        jposIntermedCentroMassa.robax.rax_4 := jposRecolhidoEsteira.robax.rax_4;
        jposIntermedCentroMassa.robax.rax_5 := jposRecolhidoEsteira.robax.rax_5;

        MoveAbsJ jposIntermedCentroMassa, sMov_Geral_Com_Produto, z200, tGarra\WObj:=wBuffer_Dir;
        GOTO inpos_fam_3;
        ENDIF

        IF (nPos_Buffer >= 1 AND nPos_Buffer <= 9) THEN
        pIntermedCentroMassa := pPosição_Final_Buffer;
	    jposIntermedCentroMassa := CalcJointT(pIntermedCentroMassa, tGarra \WObj:=wBuffer_Front);
        jposIntermedCentroMassa.robax.rax_2 := jposRecolhidoEsteira.robax.rax_2;
        jposIntermedCentroMassa.robax.rax_3 := jposRecolhidoEsteira.robax.rax_3;
        jposIntermedCentroMassa.robax.rax_4 := jposRecolhidoEsteira.robax.rax_4;
        jposIntermedCentroMassa.robax.rax_5 := jposRecolhidoEsteira.robax.rax_5;

        MoveAbsJ jposIntermedCentroMassa, sMov_Geral_Com_Produto, z200, tGarra\WObj:=wBuffer_Front;
        GOTO inpos_fam_3;
        ELSE
        pIntermedCentroMassa := pPosição_Final_Buffer;
	    jposIntermedCentroMassa := CalcJointT(pIntermedCentroMassa, tGarra \WObj:=wBuffer_Esq);
        jposIntermedCentroMassa.robax.rax_2 := jposRecolhidoEsteira.robax.rax_2;
        jposIntermedCentroMassa.robax.rax_3 := jposRecolhidoEsteira.robax.rax_3;
        jposIntermedCentroMassa.robax.rax_4 := jposRecolhidoEsteira.robax.rax_4;
        jposIntermedCentroMassa.robax.rax_5 := jposRecolhidoEsteira.robax.rax_5;

        MoveAbsJ jposIntermedCentroMassa, sMov_Geral_Com_Produto, z200, tGarra\WObj:=wBuffer_Esq;
        ENDIF

inpos_fam_3:
        !Ponto acima da posição
        pMov_Pega_Depos_Buffer := pPosição_Final_Buffer;
        pMov_Pega_Depos_Buffer.trans := pMov_Pega_Depos_Buffer.trans + pOfst_Acima_Buffer;
        IF (nPos_Buffer >= 13 AND nPos_Buffer <= 15) OR (nPos_Buffer >= 19 AND nPos_Buffer <= 21) OR (nPos_Buffer >= 25 AND nPos_Buffer <= 27) OR (nPos_Buffer >= 31 AND nPos_Buffer <=33) OR (nPos_Buffer >= 37 AND nPos_Buffer <= 39) OR (nPos_Buffer >= 43 AND nPos_Buffer <= 45) OR (nPos_Buffer >= 49 AND nPos_Buffer <= 51) OR (nPos_Buffer >= 55 AND nPos_Buffer <=57) OR (nPos_Buffer >= 61 AND nPos_Buffer <= 63) OR (nPos_Buffer >= 67 AND nPos_Buffer <= 69) OR (nPos_Buffer >= 73 AND nPos_Buffer <= 75) OR (nPos_Buffer >= 79 AND nPos_Buffer <= 81) OR (nPos_Buffer >= 85 AND nPos_Buffer <= 87) OR (nPos_Buffer >= 91 AND nPos_Buffer <= 93) OR (nPos_Buffer >= 97 AND nPos_Buffer <= 99) THEN
        MoveL pMov_Pega_Depos_Buffer, sMov_Geral_Com_Produto, fine, tGarra \WObj:=wBuffer_Dir;
        GOTO verifica_fam_3;
        ENDIF
        IF (nPos_Buffer >= 1 AND nPos_Buffer <= 9) THEN
        MoveL pMov_Pega_Depos_Buffer, sMov_Geral_Com_Produto, fine, tGarra \WObj:=wBuffer_Front;
        GOTO verifica_fam_3;
        ELSE
        MoveL pMov_Pega_Depos_Buffer, sMov_Geral_Com_Produto, fine, tGarra \WObj:=wBuffer_Esq;
        ENDIF

    verifica_fam_3:
        !Verifica se já existe peça na posição selecionada
        IF DInput (DI_Pres_Peça_Berço_1) = 0 AND DInput (DI_Pres_Peça_Berço_2) = 1 GOTO a_berço_3;

